	UF : 0, UT : 1,
	J1=   180.000 deg,	J2=   162.834 deg
};
P[215]{
   GP1:
	UF : 1, UT : 1,		CONFIG : 'N U T, 0, 0, 0',
	X =   896.264  mm,	Y =   758.406  mm,	Z =   974.529  mm,
	W =    -7.900 deg,	P =    -8.126 deg,	R =    27.442 deg
   GP2:
	UF : 0, UT : 1,
	J1=   180.000 deg,	J2=   162.834 deg
};
P[216]{
   GP1:
	UF : 1, UT : 1,		CONFIG : 'N U T, 0, 0, 0',
	X =   911.962  mm,	Y =   812.527  mm,	Z =   974.203  mm,
	W =    -6.200 deg,	P =    -4.980 deg,	R =    27.272 deg
   GP2:
	UF : 0, UT : 1,
	J1=   180.000 deg,	J2=   162.834 deg
};
P[217]{
   GP1:
	UF : 1, UT : 1,		CONFIG : 'N U T, 0, 0, 0',
	X =   899.176  mm,	Y =   819.284  mm,	Z =  1032.753  mm,
	W =     -.314 deg,	P =    -5.430 deg,	R =    27.373 deg
   GP2:
	UF : 0, UT : 1,
	J1=   180.000 deg,	J2=   162.834 deg
};
P[218]{
   GP1:
	UF : 1, UT : 1,		CONFIG : 'N U T, 0, 0, 0',
	X =   681.420  mm,	Y =   819.284  mm,	Z =  1312.752  mm,
	W =     -.314 deg,	P =    -5.430 deg,	R =    27.373 deg
   GP2:
	UF : 0, UT : 1,
	J1=   180.000 deg,	J2=   162.834 deg
};
P[219]{
   GP1:
	UF : 1, UT : 1,		CONFIG : 'N U B, 0, 0, 0',
	X =   351.047  mm,	Y =     7.833  mm,	Z =  2455.305  mm,
	W =     -.021 deg,	P =   -39.773 deg,	R =      .020 deg
   GP2:
	UF : 0, UT : 1,
	J1=   180.000 deg,	J2=   162.834 deg
};
P[220]{
   GP1:
	UF : 1, UT : 1,
	J1=     1.807 deg,	J2=   -17.141 deg,	J3=    43.457 deg,
	J4=      .157 deg,	J5=   -93.510 deg,	J6=    56.808 deg
   GP2:
	UF : 0, UT : 1,
	J1=    90.000 deg,	J2=   180.000 deg
};
P[221]{
   GP1:
	UF : 1, UT : 1,		CONFIG : 'N U T, 0, 0, 0',
	X =  1964.565  mm,	Y =     4.795  mm,	Z =  1612.445  mm,
	W =   -22.514 deg,	P =    41.901 deg,	R =    74.339 deg
   GP2:
	UF : 0, UT : 1,
	J1=    90.000 deg,	J2=   180.000 deg
};
P[222]{
   GP1:
	UF : 1, UT : 1,		CONFIG : 'N U T, 0, 0, 0',
	X =  2447.368  mm,	Y =    -1.157  mm,	Z =   875.833  mm,
	W =    -2.714 deg,	P =    44.884 deg,	R =    86.165 deg
   GP2:
	UF : 0, UT : 1,
	J1=    90.000 deg,	J2=   180.000 deg
};
P[223]{
   GP1:
	UF : 1, UT : 1,		CONFIG : 'N U T, 0, 0, 0',
	X =  2375.366  mm,	Y =   -75.636  mm,	Z =  1068.010  mm,
	W =    19.551 deg,	P =    -7.021 deg,	R =   -36.488 deg
   GP2:
	UF : 0, UT : 1,
	J1=    90.000 deg,	J2=    90.000 deg
};
P[224]{
   GP1:
	UF : 1, UT : 1,		CONFIG : 'N U T, 0, 0, 0',
	X =  2796.342  mm,	Y =  1429.156  mm,	Z =   -10.421  mm,
	W =      .000 deg,	P =      .000 deg,	R =    23.425 deg
   GP2:
	UF : 0, UT : 1,
	J1=    90.000 deg,	J2=    90.000 deg
};
P[225]{
   GP1:
	UF : 1, UT : 1,		CONFIG : 'N U T, 0, 0, 0',
	X =  2779.723  mm,	Y =  1421.979  mm,	Z =   -21.231  mm,
	W =    -1.266 deg,	P =    -3.105 deg,	R =    23.431 deg
   GP2:
	UF : 0, UT : 1,
	J1=    90.000 deg,	J2=    90.000 deg
};
P[226]{
   GP1:
	UF : 1, UT : 1,		CONFIG : 'N U T, 0, 0, 0',
	X =  2779.964  mm,	Y =  1421.713  mm,	Z =   -21.036  mm,
	W =    -1.330 deg,	P =    -3.122 deg,	R =    23.452 deg
   GP2:
	UF : 0, UT : 1,
	J1=    90.000 deg,	J2=    90.000 deg
};
P[227]{
   GP1:
	UF : 1, UT : 1,		CONFIG : 'N U T, 0, 0, 0',
	X =  2796.342  mm,	Y =  1429.156  mm,	Z =   -10.421  mm,
	W =      .000 deg,	P =      .000 deg,	R =    23.425 deg
   GP2:
	UF : 0, UT : 1,
	J1=    90.000 deg,	J2=    90.000 deg
};
P[228]{
   GP1:
	UF : 1, UT : 1,		CONFIG : 'N U T, 0, 0, 0',
	X =  2796.343  mm,	Y =  1408.935  mm,	Z =   -22.596  mm,
	W =      .000 deg,	P =      .000 deg,	R =    23.425 deg
   GP2:
	UF : 0, UT : 1,
	J1=    90.000 deg,	J2=    90.000 deg
};
P[229]{
   GP1:
	UF : 1, UT : 1,		CONFIG : 'N U T, 0, 0, 0',
	X =  2796.308  mm,	Y =  1408.958  mm,	Z =   -22.720  mm,
	W =      .007 deg,	P =      .005 deg,	R =    23.421 deg
   GP2:
	UF : 0, UT : 1,
	J1=    90.000 deg,	J2=    90.000 deg
};
P[230]{
   GP1:
	UF : 1, UT : 1,		CONFIG : 'N U T, 0, 0, 0',
	X =  2796.342  mm,	Y =  1429.156  mm,	Z =   -10.421  mm,
	W =      .000 deg,	P =      .000 deg,	R =    23.425 deg
   GP2:
	UF : 0, UT : 1,
	J1=    90.000 deg,	J2=    90.000 deg
};
P[231]{
   GP1:
	UF : 1, UT : 1,		CONFIG : 'N U T, 0, 0, 0',
	X =  2851.225  mm,	Y =  1481.272  mm,	Z =   628.377  mm,
	W =    23.286 deg,	P =   -46.577 deg,	R =   -54.612 deg
   GP2:
	UF : 0, UT : 1,
	J1=    90.000 deg,	J2=    80.000 deg
};
P[232]{
   GP1:
	UF : 1, UT : 1,		CONFIG : 'F U T, 0, 0, 0',
	X =  2809.449  mm,	Y = -1512.393  mm,	Z =   661.548  mm,
	W =   -26.535 deg,	P =   -41.775 deg,	R =    57.162 deg
   GP2:
	UF : 0, UT : 1,
	J1=    90.000 deg,	J2=   -80.000 deg
};
P[233]{
   GP1:
	UF : 1, UT : 1,		CONFIG : 'N U T, 0, 0, 0',
	X =  2141.340  mm,	Y =  -438.241  mm,	Z =   417.943  mm,
	W =   -44.721 deg,	P =     4.092 deg,	R =     4.073 deg
   GP2:
	UF : 0, UT : 1,
	J1=    89.999 deg,	J2=      .000 deg
};
P[234]{
   GP1:
	UF : 1, UT : 1,		CONFIG : 'N U T, 0, 0, 0',
	X =  2154.716  mm,	Y =  -437.126  mm,	Z =   420.005  mm,
	W =   -41.090 deg,	P =     3.840 deg,	R =     4.352 deg
   GP2:
	UF : 0, UT : 1,
	J1=    89.999 deg,	J2=      .000 deg
};
P[235]{
   GP1:
	UF : 1, UT : 1,		CONFIG : 'N U T, 0, 0, 0',
	X =  2186.155  mm,	Y =  -439.272  mm,	Z =   417.702  mm,
	W =   -40.983 deg,	P =     3.829 deg,	R =     4.326 deg
   GP2:
	UF : 0, UT : 1,
	J1=    89.999 deg,	J2=      .000 deg
};
P[236]{
   GP1:
	UF : 1, UT : 1,		CONFIG : 'N U T, 0, 0, -1',
	X =  2085.564  mm,	Y =   124.051  mm,	Z =   864.116  mm,
	W =     -.715 deg,	P =    43.124 deg,	R =   157.497 deg
   GP2:
	UF : 0, UT : 1,
	J1=    89.999 deg,	J2=    90.000 deg
};
P[672]{
   GP1:
	UF : 1, UT : 1,		CONFIG : 'N U T, 0, 0, 0',
	X =  2790.143  mm,	Y =    51.223  mm,	Z =   753.259  mm,
	W =   -32.541 deg,	P =    32.747 deg,	R =    40.290 deg
   GP2:
	UF : 0, UT : 1,
	J1=    90.000 deg,	J2=   180.000 deg
};
P[673]{
   GP1:
	UF : 1, UT : 1,		CONFIG : 'N U T, 0, 0, 0',
	X =  2827.690  mm,	Y =    49.321  mm,	Z =   754.374  mm,
	W =   -32.607 deg,	P =    32.790 deg,	R =    40.253 deg
   GP2:
	UF : 0, UT : 1,
	J1=    90.000 deg,	J2=   180.000 deg
};
P[674]{
   GP1:
	UF : 1, UT : 1,		CONFIG : 'N U T, 0, 0, 0',
	X =  2780.720  mm,	Y =    85.310  mm,	Z =   845.034  mm,
	W =   -26.000 deg,	P =    27.653 deg,	R =    43.586 deg
   GP2:
	UF : 0, UT : 1,
	J1=    90.000 deg,	J2=   180.000 deg
};
P[675]{
   GP1:
	UF : 1, UT : 1,		CONFIG : 'N U T, 0, 0, 0',
	X =  2810.125  mm,	Y =   -14.508  mm,	Z =   877.692  mm,
	W =     4.233 deg,	P =     1.150 deg,	R =   -15.151 deg
   GP2:
	UF : 0, UT : 1,
	J1=    90.000 deg,	J2=   180.000 deg
};
P[676]{
   GP1:
	UF : 1, UT : 1,		CONFIG : 'N U T, 0, 0, 0',
	X =  2779.721  mm,	Y =   -75.691  mm,	Z =   818.586  mm,
	W =    22.126 deg,	P =    31.326 deg,	R =   -51.965 deg
   GP2:
	UF : 0, UT : 1,
	J1=    90.000 deg,	J2=   180.000 deg
};
P[677]{
   GP1:
	UF : 1, UT : 1,		CONFIG : 'N U T, 0, 0, 0',
	X =  2792.677  mm,	Y =   -55.688  mm,	Z =   756.492  mm,
	W =    24.186 deg,	P =    33.500 deg,	R =   -50.860 deg
   GP2:
	UF : 0, UT : 1,
	J1=    90.000 deg,	J2=   180.000 deg
};
P[678]{
   GP1:
	UF : 1, UT : 1,		CONFIG : 'N U T, 0, 0, 0',
	X =  2832.302  mm,	Y =   -54.185  mm,	Z =   758.283  mm,
	W =    24.209 deg,	P =    33.526 deg,	R =   -50.852 deg
   GP2:
	UF : 0, UT : 1,
	J1=    90.000 deg,	J2=   180.000 deg
};
P[679]{
   GP1:
	UF : 1, UT : 1,		CONFIG : 'N U T, 0, 0, 0',
	X =  2779.721  mm,	Y =   -75.691  mm,	Z =   876.586  mm,
	W =    23.118 deg,	P =    32.394 deg,	R =   -51.441 deg
   GP2:
	UF : 0, UT : 1,
	J1=    90.000 deg,	J2=   180.000 deg
};
P[680]{
   GP1:
	UF : 1, UT : 1,		CONFIG : 'N U T, 0, 0, 0',
	X =  2779.721  mm,	Y =   -75.691  mm,	Z =   876.586  mm,
	W =     -.000 deg,	P =     6.847 deg,	R =      .007 deg
   GP2:
	UF : 0, UT : 1,
	J1=    90.000 deg,	J2=   180.000 deg
};
P[681]{
   GP1:
	UF : 1, UT : 1,		CONFIG : 'N U T, 0, 0, 0',
	X =  2840.099  mm,	Y =   -54.094  mm,	Z =   811.805  mm,
	W =      .000 deg,	P =    10.475 deg,	R =      .007 deg
   GP2:
	UF : 0, UT : 1,
	J1=    90.000 deg,	J2=   180.000 deg
};
P[682]{
   GP1:
	UF : 1, UT : 1,		CONFIG : 'N U T, 0, 0, 0',
	X =  2840.358  mm,	Y =   -49.439  mm,	Z =   753.835  mm,
	W =      .034 deg,	P =    10.479 deg,	R =      .019 deg
   GP2:
	UF : 0, UT : 1,
	J1=    90.000 deg,	J2=   180.000 deg
};
P[683]{
   GP1:
	UF : 1, UT : 1,		CONFIG : 'N U T, 0, 0, 0',
	X =  2841.066  mm,	Y =    46.936  mm,	Z =   753.793  mm,
	W =      .058 deg,	P =    10.474 deg,	R =      .009 deg
   GP2:
	UF : 0, UT : 1,
	J1=    90.000 deg,	J2=   180.000 deg
};
P[684]{
   GP1:
	UF : 1, UT : 1,		CONFIG : 'N U T, 0, 0, 0',
	X =  2840.099  mm,	Y =   -54.094  mm,	Z =   811.805  mm,
	W =      .000 deg,	P =    10.475 deg,	R =      .007 deg
   GP2:
	UF : 0, UT : 1,
	J1=    90.000 deg,	J2=   180.000 deg
};
P[685]{
   GP1:
	UF : 1, UT : 1,		CONFIG : 'N U T, 0, 0, 0',
	X =  2685.813  mm,	Y =   -54.094  mm,	Z =  1008.948  mm,
	W =     -.002 deg,	P =   -13.112 deg,	R =      .007 deg
   GP2:
	UF : 0, UT : 1,
	J1=    90.000 deg,	J2=   180.000 deg
};
P[686]{
   GP1:
	UF : 1, UT : 1,		CONFIG : 'N U T, 0, 0, 0',
	X =  1792.252  mm,	Y =    19.310  mm,	Z =   722.821  mm,
	W =   -31.232 deg,	P =    38.925 deg,	R =    72.124 deg
   GP2:
	UF : 0, UT : 1,
	J1=    90.000 deg,	J2=   180.000 deg
};
P[687]{
   GP1:
	UF : 1, UT : 1,		CONFIG : 'N U T, 0, 0, 0',
	X =  1696.704  mm,	Y =  -379.767  mm,	Z =   546.319  mm,
	W =     0.000 deg,	P =    43.571 deg,	R =    90.007 deg
   GP2:
	UF : 0, UT : 1,
	J1=    90.000 deg,	J2=   180.000 deg
};
P[688]{
   GP1:
	UF : 1, UT : 1,		CONFIG : 'N U T, 0, 0, 0',
	X =  1720.777  mm,	Y =  -450.296  mm,	Z =   422.624  mm,
	W =     -.005 deg,	P =    43.535 deg,	R =    86.286 deg
   GP2:
	UF : 0, UT : 1,
	J1=    90.000 deg,	J2=   180.000 deg
};
P[689]{
   GP1:
	UF : 1, UT : 1,		CONFIG : 'N U T, 0, 0, 0',
	X =  1580.851  mm,	Y =  -449.343  mm,	Z =   421.313  mm,
	W =     -.007 deg,	P =    43.521 deg,	R =    86.268 deg
   GP2:
	UF : 0, UT : 1,
	J1=    90.000 deg,	J2=   180.000 deg
};
P[690]{
   GP1:
	UF : 1, UT : 1,		CONFIG : 'N U T, 0, 0, 0',
	X =  1587.135  mm,	Y =  -378.521  mm,	Z =   501.393  mm,
	W =      .000 deg,	P =    43.571 deg,	R =    86.288 deg
   GP2:
	UF : 0, UT : 1,
	J1=    90.000 deg,	J2=   180.000 deg
};
P[691]{
   GP1:
	UF : 1, UT : 1,		CONFIG : 'N U T, 0, 0, 0',
	X =  1998.349  mm,	Y =  -373.244  mm,	Z =   510.901  mm,
	W =   -38.646 deg,	P =    21.930 deg,	R =    21.323 deg
   GP2:
	UF : 0, UT : 1,
	J1=    90.000 deg,	J2=   180.000 deg
};
P[692]{
   GP1:
	UF : 1, UT : 1,		CONFIG : 'N U T, 0, 0, 0',
	X =  1957.677  mm,	Y =  -448.116  mm,	Z =   422.495  mm,
	W =   -40.835 deg,	P =    20.797 deg,	R =    22.335 deg
   GP2:
	UF : 0, UT : 1,
	J1=    90.000 deg,	J2=   180.000 deg
};
P[693]{
   GP1:
	UF : 1, UT : 1,		CONFIG : 'N U T, 0, 0, 0',
	X =  2027.930  mm,	Y =  -449.856  mm,	Z =   421.404  mm,
	W =   -43.530 deg,	P =    18.886 deg,	R =    21.391 deg
   GP2:
	UF : 0, UT : 1,
	J1=    90.000 deg,	J2=   180.000 deg
};
P[694]{
   GP1:
	UF : 1, UT : 1,		CONFIG : 'N U T, 0, 0, 0',
	X =  2047.306  mm,	Y =  -108.854  mm,	Z =   590.153  mm,
	W =   -38.646 deg,	P =    21.930 deg,	R =    21.323 deg
   GP2:
	UF : 0, UT : 1,
	J1=    90.000 deg,	J2=   180.000 deg
};
P[695]{
   GP1:
	UF : 1, UT : 1,		CONFIG : 'N U T, 0, 0, 0',
	X =  2053.592  mm,	Y =  -292.854  mm,	Z =   563.211  mm,
	W =   -43.351 deg,	P =    -4.892 deg,	R =    40.339 deg
   GP2:
	UF : 0, UT : 1,
	J1=    90.000 deg,	J2=   180.000 deg
};
P[696]{
   GP1:
	UF : 1, UT : 1,		CONFIG : 'N U T, 0, 0, 0',
	X =  2144.764  mm,	Y =  -384.746  mm,	Z =   419.107  mm,
	W =   -44.891 deg,	P =    -3.592 deg,	R =    39.096 deg
   GP2:
	UF : 0, UT : 1,
	J1=    90.000 deg,	J2=   180.000 deg
};
P[697]{
   GP1:
	UF : 1, UT : 1,		CONFIG : 'N U T, 0, 0, 0',
	X =  2100.455  mm,	Y =  -424.853  mm,	Z =   417.888  mm,
	W =   -43.231 deg,	P =    13.871 deg,	R =    57.009 deg
   GP2:
	UF : 0, UT : 1,
	J1=    89.999 deg,	J2=   180.000 deg
};
P[698]{
   GP1:
	UF : 1, UT : 1,		CONFIG : 'N U T, 0, 0, 0',
	X =  2099.808  mm,	Y =  -430.674  mm,	Z =   419.684  mm,
	W =   -44.233 deg,	P =    -9.263 deg,	R =    60.679 deg
   GP2:
	UF : 0, UT : 1,
	J1=    89.999 deg,	J2=   180.000 deg
};
P[699]{
   GP1:
	UF : 1, UT : 1,		CONFIG : 'N U T, 0, 0, 0',
	X =  2096.561  mm,	Y =  -436.435  mm,	Z =   421.890  mm,
	W =   -46.555 deg,	P =    -2.361 deg,	R =    62.902 deg
   GP2:
	UF : 0, UT : 1,
	J1=    90.000 deg,	J2=   180.000 deg
};
P[700]{
   GP1:
	UF : 1, UT : 1,		CONFIG : 'N U T, 0, 0, 0',
	X =  1980.139  mm,	Y =  -394.363  mm,	Z =   568.863  mm,
	W =   -43.468 deg,	P =    -3.333 deg,	R =    66.484 deg
   GP2:
	UF : 0, UT : 1,
	J1=    90.000 deg,	J2=   180.000 deg
};
P[701]{
   GP1:
	UF : 1, UT : 1,		CONFIG : 'N U T, 0, 0, 0',
	X =  1759.952  mm,	Y =   241.660  mm,	Z =   616.315  mm,
	W =    29.266 deg,	P =    41.264 deg,	R =   -11.299 deg
   GP2:
	UF : 0, UT : 1,
	J1=    90.000 deg,	J2=   180.000 deg
};
P[702]{
   GP1:
	UF : 1, UT : 1,		CONFIG : 'N U T, 0, 0, 0',
	X =  1720.918  mm,	Y =   388.510  mm,	Z =   489.828  mm,
	W =     0.000 deg,	P =    43.571 deg,	R =   -89.993 deg
   GP2:
	UF : 0, UT : 1,
	J1=    90.000 deg,	J2=   180.000 deg
};
P[703]{
   GP1:
	UF : 1, UT : 1,		CONFIG : 'N U T, 0, 0, 0',
	X =  1722.929  mm,	Y =   446.414  mm,	Z =   421.655  mm,
	W =    -1.651 deg,	P =    44.983 deg,	R =   -92.337 deg
   GP2:
	UF : 0, UT : 1,
	J1=    90.000 deg,	J2=   180.000 deg
};
P[704]{
   GP1:
	UF : 1, UT : 1,		CONFIG : 'N U T, 0, 0, 0',
	X =  1584.785  mm,	Y =   445.500  mm,	Z =   419.176  mm,
	W =    -1.657 deg,	P =    45.006 deg,	R =   -92.336 deg
   GP2:
	UF : 0, UT : 1,
	J1=    90.000 deg,	J2=   180.000 deg
};
P[705]{
   GP1:
	UF : 1, UT : 1,		CONFIG : 'N U T, 0, 0, 0',
	X =  1594.524  mm,	Y =   351.963  mm,	Z =   523.980  mm,
	W =      .000 deg,	P =    43.571 deg,	R =   -92.306 deg
   GP2:
	UF : 0, UT : 1,
	J1=    90.000 deg,	J2=   180.000 deg
};
P[706]{
   GP1:
	UF : 1, UT : 1,		CONFIG : 'N U T, 0, 0, 0',
	X =  1972.524  mm,	Y =   351.963  mm,	Z =   523.980  mm,
	W =    31.879 deg,	P =    31.438 deg,	R =   -42.291 deg
   GP2:
	UF : 0, UT : 1,
	J1=    90.000 deg,	J2=   180.000 deg
};
P[707]{
   GP1:
	UF : 1, UT : 1,		CONFIG : 'N U T, 0, 0, 0',
	X =  1957.584  mm,	Y =   447.653  mm,	Z =   420.327  mm,
	W =    32.281 deg,	P =    33.246 deg,	R =   -40.947 deg
   GP2:
	UF : 0, UT : 1,
	J1=    90.000 deg,	J2=   180.000 deg
};
P[708]{
   GP1:
	UF : 1, UT : 1,		CONFIG : 'N U T, 0, 0, 0',
	X =  2031.416  mm,	Y =   447.860  mm,	Z =   420.354  mm,
	W =    34.389 deg,	P =    31.198 deg,	R =   -39.833 deg
   GP2:
	UF : 0, UT : 1,
	J1=    90.000 deg,	J2=   180.000 deg
};
P[709]{
   GP1:
	UF : 1, UT : 1,		CONFIG : 'N U T, 0, 0, 0',
	X =  2028.229  mm,	Y =   306.190  mm,	Z =   574.407  mm,
	W =    39.948 deg,	P =    19.080 deg,	R =   -23.626 deg
   GP2:
	UF : 0, UT : 1,
	J1=    90.000 deg,	J2=   180.000 deg
};
P[710]{
   GP1:
	UF : 1, UT : 1,		CONFIG : 'N U T, 0, 0, 0',
	X =  2028.228  mm,	Y =   306.190  mm,	Z =   574.407  mm,
	W =    39.948 deg,	P =    19.080 deg,	R =   -73.748 deg
   GP2:
	UF : 0, UT : 1,
	J1=    90.000 deg,	J2=   180.000 deg
};
P[711]{
   GP1:
	UF : 1, UT : 1,		CONFIG : 'N U T, 0, 0, 0',
	X =  2146.185  mm,	Y =   382.939  mm,	Z =   421.328  mm,
	W =    42.385 deg,	P =    16.872 deg,	R =   -60.307 deg
   GP2:
	UF : 0, UT : 1,
	J1=    90.000 deg,	J2=   180.000 deg
};
P[712]{
   GP1:
	UF : 1, UT : 1,		CONFIG : 'N U T, 0, 0, 0',
	X =  2104.195  mm,	Y =   420.889  mm,	Z =   422.475  mm,
	W =    44.151 deg,	P =     9.880 deg,	R =   -52.687 deg
   GP2:
	UF : 0, UT : 1,
	J1=    90.000 deg,	J2=   180.000 deg
};
P[713]{
   GP1:
	UF : 1, UT : 1,		CONFIG : 'N U T, 0, 0, 0',
	X =  2101.951  mm,	Y =   428.282  mm,	Z =   420.792  mm,
	W =    44.777 deg,	P =    -5.046 deg,	R =   -67.249 deg
   GP2:
	UF : 0, UT : 1,
	J1=    89.999 deg,	J2=   180.000 deg
};
P[714]{
   GP1:
	UF : 1, UT : 1,		CONFIG : 'N U T, 0, 0, 0',
	X =  2101.615  mm,	Y =   433.364  mm,	Z =   421.849  mm,
	W =    42.053 deg,	P =   -17.708 deg,	R =   -50.532 deg
   GP2:
	UF : 0, UT : 1,
	J1=    89.999 deg,	J2=   180.000 deg
};
P[715]{
   GP1:
	UF : 1, UT : 1,		CONFIG : 'N U T, 0, 0, 0',
	X =  2002.025  mm,	Y =   135.053  mm,	Z =   547.724  mm,
	W =    43.132 deg,	P =    -6.887 deg,	R =   -61.237 deg
   GP2:
	UF : 0, UT : 1,
	J1=    90.000 deg,	J2=   180.000 deg
};
P[716]{
   GP1:
	UF : 1, UT : 1,		CONFIG : 'N U T, 0, 0, 0',
	X =  2377.025  mm,	Y =   240.053  mm,	Z =   291.724  mm,
	W =    40.241 deg,	P =    18.349 deg,	R =   -20.268 deg
   GP2:
	UF : 0, UT : 1,
	J1=    90.000 deg,	J2=   180.000 deg
};
P[717]{
   GP1:
	UF : 1, UT : 1,		CONFIG : 'N U T, 0, 0, 0',
	X =  2355.551  mm,	Y =   374.115  mm,	Z =   302.484  mm,
	W =    40.241 deg,	P =    18.349 deg,	R =   -20.268 deg
   GP2:
	UF : 0, UT : 1,
	J1=    90.000 deg,	J2=   180.000 deg
};
P[718]{
   GP1:
	UF : 1, UT : 1,		CONFIG : 'N U T, 0, 0, 0',
	X =  2349.451  mm,	Y =   438.430  mm,	Z =   272.108  mm,
	W =    44.913 deg,	P =     3.071 deg,	R =    -3.074 deg
   GP2:
	UF : 0, UT : 1,
	J1=    90.000 deg,	J2=   180.000 deg
};
P[719]{
   GP1:
	UF : 1, UT : 1,		CONFIG : 'N U T, 0, 0, 0',
	X =  2407.584  mm,	Y =   438.337  mm,	Z =   273.841  mm,
	W =    38.958 deg,	P =   -20.279 deg,	R =    -1.908 deg
   GP2:
	UF : 0, UT : 1,
	J1=    89.999 deg,	J2=   180.000 deg
};
P[720]{
   GP1:
	UF : 1, UT : 1,		CONFIG : 'N U T, 0, 0, 0',
	X =  2355.551  mm,	Y =   374.115  mm,	Z =   302.484  mm,
	W =    40.241 deg,	P =    18.349 deg,	R =   -20.268 deg
   GP2:
	UF : 0, UT : 1,
	J1=    90.000 deg,	J2=   180.000 deg
};
P[721]{
   GP1:
	UF : 1, UT : 1,		CONFIG : 'N U T, 0, 0, 0',
	X =  2355.551  mm,	Y =   222.115  mm,	Z =   302.484  mm,
	W =    40.242 deg,	P =    18.350 deg,	R =   -20.267 deg
   GP2:
	UF : 0, UT : 1,
	J1=    90.000 deg,	J2=   180.000 deg
};
P[722]{
   GP1:
	UF : 1, UT : 1,		CONFIG : 'N U T, 0, 0, 0',
	X =  2484.503  mm,	Y =   222.115  mm,	Z =   302.484  mm,
	W =    43.394 deg,	P =    -4.399 deg,	R =     4.775 deg
   GP2:
	UF : 0, UT : 1,
	J1=    90.000 deg,	J2=   180.000 deg
};
P[723]{
   GP1:
	UF : 1, UT : 1,		CONFIG : 'N U T, 0, 0, 0',
	X =  2484.503  mm,	Y =   285.115  mm,	Z =   258.737  mm,
	W =    43.394 deg,	P =    -4.398 deg,	R =     4.776 deg
   GP2:
	UF : 0, UT : 1,
	J1=    90.000 deg,	J2=   180.000 deg
};
P[724]{
   GP1:
	UF : 1, UT : 1,		CONFIG : 'N U T, 0, 0, 0',
	X =  2482.396  mm,	Y =   435.010  mm,	Z =   224.036  mm,
	W =     9.249 deg,	P =   -44.227 deg,	R =    76.876 deg
   GP2:
	UF : 0, UT : 1,
	J1=    90.000 deg,	J2=   180.000 deg
};
P[725]{
   GP1:
	UF : 1, UT : 1,		CONFIG : 'N U T, 0, 0, 0',
	X =  2430.889  mm,	Y =   433.696  mm,	Z =   223.972  mm,
	W =    35.355 deg,	P =   -42.180 deg,	R =    70.882 deg
   GP2:
	UF : 0, UT : 1,
	J1=    90.000 deg,	J2=   180.000 deg
};
P[726]{
   GP1:
	UF : 1, UT : 1,		CONFIG : 'N U T, 0, 0, 0',
	X =  2484.503  mm,	Y =   285.115  mm,	Z =   258.737  mm,
	W =    43.394 deg,	P =    -4.398 deg,	R =     4.776 deg
   GP2:
	UF : 0, UT : 1,
	J1=    90.000 deg,	J2=   180.000 deg
};
P[727]{
   GP1:
	UF : 1, UT : 1,		CONFIG : 'N U T, 0, 0, 0',
	X =  2484.503  mm,	Y =   222.115  mm,	Z =   302.485  mm,
	W =    43.394 deg,	P =    -4.399 deg,	R =     4.775 deg
   GP2:
	UF : 0, UT : 1,
	J1=    90.000 deg,	J2=   180.000 deg
};
P[728]{
   GP1:
	UF : 1, UT : 1,		CONFIG : 'N U T, 0, 0, 0',
	X =  2355.551  mm,	Y =     2.115  mm,	Z =   302.485  mm,
	W =     5.759 deg,	P =    43.266 deg,	R =    98.508 deg
   GP2:
	UF : 0, UT : 1,
	J1=    90.000 deg,	J2=   180.000 deg
};
P[729]{
   GP1:
	UF : 1, UT : 1,		CONFIG : 'N U T, 0, 0, 0',
	X =  2355.551  mm,	Y =  -363.653  mm,	Z =   302.484  mm,
	W =   -43.559 deg,	P =     1.197 deg,	R =     1.395 deg
   GP2:
	UF : 0, UT : 1,
	J1=    90.000 deg,	J2=   180.000 deg
};
P[730]{
   GP1:
	UF : 1, UT : 1,		CONFIG : 'N U T, 0, 0, 0',
	X =  2346.935  mm,	Y =  -439.624  mm,	Z =   272.632  mm,
	W =   -44.978 deg,	P =     1.293 deg,	R =     1.297 deg
   GP2:
	UF : 0, UT : 1,
	J1=    90.000 deg,	J2=   180.000 deg
};
P[731]{
   GP1:
	UF : 1, UT : 1,		CONFIG : 'N U T, 0, 0, 0',
	X =  2407.646  mm,	Y =  -437.669  mm,	Z =   274.279  mm,
	W =   -45.256 deg,	P =   -24.481 deg,	R =     5.929 deg
   GP2:
	UF : 0, UT : 1,
	J1=    89.999 deg,	J2=   180.000 deg
};
P[732]{
   GP1:
	UF : 1, UT : 1,		CONFIG : 'N U T, 0, 0, 0',
	X =  2355.551  mm,	Y =  -363.653  mm,	Z =   302.484  mm,
	W =   -43.559 deg,	P =     1.197 deg,	R =     1.395 deg
   GP2:
	UF : 0, UT : 1,
	J1=    90.000 deg,	J2=   180.000 deg
};
P[733]{
   GP1:
	UF : 1, UT : 1,		CONFIG : 'N U T, 0, 0, 0',
	X =  2355.551  mm,	Y =  -226.653  mm,	Z =   302.484  mm,
	W =   -43.560 deg,	P =     1.197 deg,	R =     1.395 deg
   GP2:
	UF : 0, UT : 1,
	J1=    90.000 deg,	J2=   180.000 deg
};
P[734]{
   GP1:
	UF : 1, UT : 1,		CONFIG : 'N U T, 0, 0, 0',
	X =  2475.388  mm,	Y =  -226.653  mm,	Z =   302.484  mm,
	W =   -29.446 deg,	P =   -33.698 deg,	R =   -44.366 deg
   GP2:
	UF : 0, UT : 1,
	J1=    90.000 deg,	J2=   180.000 deg
};
P[735]{
   GP1:
	UF : 1, UT : 1,		CONFIG : 'N U T, 0, 0, 0',
	X =  2484.256  mm,	Y =  -439.439  mm,	Z =   222.852  mm,
	W =    -2.387 deg,	P =   -44.924 deg,	R =   -86.621 deg
   GP2:
	UF : 0, UT : 1,
	J1=    90.000 deg,	J2=   180.000 deg
};
P[736]{
   GP1:
	UF : 1, UT : 1,		CONFIG : 'N U T, 0, 0, 0',
	X =  2426.375  mm,	Y =  -437.302  mm,	Z =   225.413  mm,
	W =   -26.791 deg,	P =   -43.570 deg,	R =   -86.675 deg
   GP2:
	UF : 0, UT : 1,
	J1=    90.000 deg,	J2=   180.000 deg
};
P[737]{
   GP1:
	UF : 1, UT : 1,		CONFIG : 'N U T, 0, 0, 0',
	X =  2475.389  mm,	Y =  -226.653  mm,	Z =   302.484  mm,
	W =   -29.446 deg,	P =   -33.698 deg,	R =   -44.366 deg
   GP2:
	UF : 0, UT : 1,
	J1=    90.000 deg,	J2=   180.000 deg
};
P[738]{
   GP1:
	UF : 1, UT : 1,		CONFIG : 'N U T, 0, 0, 0',
	X =  2475.361  mm,	Y =  -127.379  mm,	Z =   161.610  mm,
	W =    -9.376 deg,	P =    15.683 deg,	R =   -16.267 deg
   GP2:
	UF : 0, UT : 1,
	J1=    90.000 deg,	J2=   180.000 deg
};
P[739]{
   GP1:
	UF : 1, UT : 1,		CONFIG : 'N U T, 0, 0, 0',
	X =  2184.132  mm,	Y =   -42.626  mm,	Z =   871.946  mm,
	W =    -9.375 deg,	P =    15.689 deg,	R =   -16.266 deg
   GP2:
	UF : 0, UT : 1,
	J1=    90.000 deg,	J2=   180.000 deg
};
P[740]{
   GP1:
	UF : 1, UT : 1,		CONFIG : 'N U B, 0, 0, 0',
	X =   390.614  mm,	Y =     -.024  mm,	Z =  2434.016  mm,
	W =     -.021 deg,	P =   -39.773 deg,	R =      .020 deg
   GP2:
	UF : 0, UT : 1,
	J1=    90.000 deg,	J2=   180.000 deg
};
P[741]{
   GP1:
	UF : 1, UT : 1,
	J1=     -.065 deg,	J2=   -43.813 deg,	J3=    64.455 deg,
	J4=     -.068 deg,	J5=   -69.455 deg,	J6=      .029 deg
   GP2:
	UF : 0, UT : 1,
	J1=    90.000 deg,	J2=     0.000 deg
};
P[742]{
   GP1:
	UF : 1, UT : 1,		CONFIG : 'N U T, 0, 0, 0',
	X =  1852.631  mm,	Y =    -6.774  mm,	Z =   565.209  mm,
	W =     -.000 deg,	P =    45.917 deg,	R =    -2.669 deg
   GP2:
	UF : 0, UT : 1,
	J1=    90.000 deg,	J2=     0.000 deg
};
P[743]{
   GP1:
	UF : 1, UT : 1,		CONFIG : 'N U T, 0, 0, 0',
	X =  1655.504  mm,	Y =   141.226  mm,	Z =   511.209  mm,
	W =     -.000 deg,	P =    45.917 deg,	R =    -2.669 deg
   GP2:
	UF : 0, UT : 1,
	J1=    90.000 deg,	J2=     0.000 deg
};
P[744]{
   GP1:
	UF : 1, UT : 1,		CONFIG : 'N U T, 0, 0, 0',
	X =  1609.671  mm,	Y =   144.502  mm,	Z =   412.787  mm,
	W =      .173 deg,	P =    45.931 deg,	R =    -2.572 deg
   GP2:
	UF : 0, UT : 1,
	J1=    90.000 deg,	J2=     -.000 deg
};
P[745]{
   GP1:
	UF : 1, UT : 1,		CONFIG : 'N U T, 0, 0, 0',
	X =  1610.947  mm,	Y =   248.052  mm,	Z =   413.254  mm,
	W =      .102 deg,	P =    45.934 deg,	R =    -2.609 deg
   GP2:
	UF : 0, UT : 1,
	J1=    89.999 deg,	J2=      .000 deg
};
P[746]{
   GP1:
	UF : 1, UT : 1,		CONFIG : 'N U T, 0, 0, 0',
	X =  1637.136  mm,	Y =   314.793  mm,	Z =   459.534  mm,
	W =     -.000 deg,	P =    45.917 deg,	R =    -2.669 deg
   GP2:
	UF : 0, UT : 1,
	J1=    90.000 deg,	J2=     0.000 deg
};
P[747]{
   GP1:
	UF : 1, UT : 1,		CONFIG : 'N U T, 0, 0, 0',
	X =  1612.461  mm,	Y =   348.792  mm,	Z =   411.820  mm,
	W =    -2.031 deg,	P =    48.815 deg,	R =    -2.770 deg
   GP2:
	UF : 0, UT : 1,
	J1=    89.999 deg,	J2=      .000 deg
};
P[748]{
   GP1:
	UF : 1, UT : 1,		CONFIG : 'N U T, 0, 0, 0',
	X =  1610.257  mm,	Y =   432.690  mm,	Z =   411.364  mm,
	W =    32.767 deg,	P =    34.177 deg,	R =    46.223 deg
   GP2:
	UF : 0, UT : 1,
	J1=    90.000 deg,	J2=      .000 deg
};
P[749]{
   GP1:
	UF : 1, UT : 1,		CONFIG : 'N U T, 0, 0, 0',
	X =  1691.137  mm,	Y =   314.793  mm,	Z =   549.534  mm,
	W =     -.000 deg,	P =    45.918 deg,	R =    -2.669 deg
   GP2:
	UF : 0, UT : 1,
	J1=    90.000 deg,	J2=     0.000 deg
};
P[750]{
   GP1:
	UF : 1, UT : 1,		CONFIG : 'N U T, 0, 0, 0',
	X =  1691.136  mm,	Y =  -139.207  mm,	Z =   549.534  mm,
	W =     -.000 deg,	P =    45.919 deg,	R =    -2.669 deg
   GP2:
	UF : 0, UT : 1,
	J1=    90.000 deg,	J2=     0.000 deg
};
P[751]{
   GP1:
	UF : 1, UT : 1,		CONFIG : 'N U T, 0, 0, 0',
	X =  1611.466  mm,	Y =  -130.160  mm,	Z =   407.191  mm,
	W =      .132 deg,	P =    45.900 deg,	R =    -2.610 deg
   GP2:
	UF : 0, UT : 1,
	J1=    89.999 deg,	J2=      .000 deg
};
P[752]{
   GP1:
	UF : 1, UT : 1,		CONFIG : 'N U T, 0, 0, 0',
	X =  1612.455  mm,	Y =  -157.655  mm,	Z =   408.458  mm,
	W =      .071 deg,	P =    45.910 deg,	R =    -2.628 deg
   GP2:
	UF : 0, UT : 1,
	J1=    90.000 deg,	J2=      .000 deg
};
P[753]{
   GP1:
	UF : 1, UT : 1,		CONFIG : 'N U T, 0, 0, 0',
	X =  1701.553  mm,	Y =  -162.044  mm,	Z =   513.926  mm,
	W =      .001 deg,	P =    45.916 deg,	R =    -2.666 deg
   GP2:
	UF : 0, UT : 1,
	J1=    90.000 deg,	J2=     0.000 deg
};
P[754]{
   GP1:
	UF : 1, UT : 1,		CONFIG : 'N U T, 0, 0, 0',
	X =  1651.458  mm,	Y =  -207.923  mm,	Z =   466.756  mm,
	W =      .001 deg,	P =    45.916 deg,	R =    15.512 deg
   GP2:
	UF : 0, UT : 1,
	J1=    90.000 deg,	J2=     0.000 deg
};
P[755]{
   GP1:
	UF : 1, UT : 1,		CONFIG : 'N U T, 0, 0, 0',
	X =  1611.664  mm,	Y =  -223.720  mm,	Z =   410.590  mm,
	W =    -1.058 deg,	P =    39.466 deg,	R =    14.834 deg
   GP2:
	UF : 0, UT : 1,
	J1=    90.000 deg,	J2=      .000 deg
};
P[756]{
   GP1:
	UF : 1, UT : 1,		CONFIG : 'N U T, 0, 0, 0',
	X =  1613.255  mm,	Y =  -156.646  mm,	Z =   408.642  mm,
	W =     3.854 deg,	P =    34.718 deg,	R =   -21.298 deg
   GP2:
	UF : 0, UT : 1,
	J1=    90.000 deg,	J2=      .000 deg
};
P[757]{
   GP1:
	UF : 1, UT : 1,		CONFIG : 'N U T, 0, 0, 0',
	X =  1663.438  mm,	Y =  -190.775  mm,	Z =   486.236  mm,
	W =      .001 deg,	P =    45.916 deg,	R =   -32.606 deg
   GP2:
	UF : 0, UT : 1,
	J1=    90.000 deg,	J2=     0.000 deg
};
P[758]{
   GP1:
	UF : 1, UT : 1,		CONFIG : 'N U T, 0, 0, 0',
	X =  1694.246  mm,	Y =  -335.221  mm,	Z =   519.016  mm,
	W =   -24.937 deg,	P =    39.897 deg,	R =   -38.608 deg
   GP2:
	UF : 0, UT : 1,
	J1=    90.000 deg,	J2=     0.000 deg
};
P[759]{
   GP1:
	UF : 1, UT : 1,		CONFIG : 'N U T, 0, 0, 0',
	X =  1609.958  mm,	Y =  -354.596  mm,	Z =   409.981  mm,
	W =   -28.732 deg,	P =    41.555 deg,	R =   -39.650 deg
   GP2:
	UF : 0, UT : 1,
	J1=    90.000 deg,	J2=      .000 deg
};
P[760]{
   GP1:
	UF : 1, UT : 1,		CONFIG : 'N U T, 0, 0, 0',
	X =  1607.480  mm,	Y =  -434.366  mm,	Z =   408.044  mm,
	W =   -34.474 deg,	P =    37.257 deg,	R =   -48.669 deg
   GP2:
	UF : 0, UT : 1,
	J1=    90.000 deg,	J2=      .000 deg
};
P[761]{
   GP1:
	UF : 1, UT : 1,		CONFIG : 'N U T, 0, 0, 0',
	X =  1714.229  mm,	Y =  -410.520  mm,	Z =   541.553  mm,
	W =   -30.592 deg,	P =    36.083 deg,	R =   -32.808 deg
   GP2:
	UF : 0, UT : 1,
	J1=    90.000 deg,	J2=     0.000 deg
};
P[762]{
   GP1:
	UF : 1, UT : 1,		CONFIG : 'N U T, 0, 0, 0',
	X =  1852.631  mm,	Y =    -6.774  mm,	Z =   565.209  mm,
	W =     -.000 deg,	P =    45.917 deg,	R =    -2.669 deg
   GP2:
	UF : 0, UT : 1,
	J1=    90.000 deg,	J2=     0.000 deg
};
P[763]{
   GP1:
	UF : 1, UT : 1,		CONFIG : 'N U T, 0, 0, 0',
	X =  2052.631  mm,	Y =  -276.774  mm,	Z =   565.209  mm,
	W =   -41.084 deg,	P =    22.633 deg,	R =    21.147 deg
   GP2:
	UF : 0, UT : 1,
	J1=    90.000 deg,	J2=     0.000 deg
};
P[764]{
   GP1:
	UF : 1, UT : 1,		CONFIG : 'N U T, 0, 0, 0',
	X =  2088.553  mm,	Y =  -373.284  mm,	Z =   491.208  mm,
	W =   -45.800 deg,	P =     3.716 deg,	R =      .937 deg
   GP2:
	UF : 0, UT : 1,
	J1=    90.000 deg,	J2=     0.000 deg
};
P[765]{
   GP1:
	UF : 1, UT : 1,		CONFIG : 'N U T, 0, 0, 0',
	X =  2063.471  mm,	Y =  -440.130  mm,	Z =   414.294  mm,
	W =   -44.841 deg,	P =     4.112 deg,	R =     4.121 deg
   GP2:
	UF : 0, UT : 1,
	J1=    90.000 deg,	J2=      .000 deg
};
P[766]{
   GP1:
	UF : 1, UT : 1,		CONFIG : 'N U T, 0, 0, 0',
	X =  2311.826  mm,	Y =  -442.485  mm,	Z =   415.387  mm,
	W =   -44.797 deg,	P =     4.102 deg,	R =     4.097 deg
   GP2:
	UF : 0, UT : 1,
	J1=    89.999 deg,	J2=      .000 deg
};
P[767]{
   GP1:
	UF : 1, UT : 1,		CONFIG : 'N U T, 0, 0, 0',
	X =  2305.976  mm,	Y =  -368.534  mm,	Z =   500.330  mm,
	W =   -45.801 deg,	P =     3.717 deg,	R =     4.521 deg
   GP2:
	UF : 0, UT : 1,
	J1=    90.000 deg,	J2=     0.000 deg
};
P[768]{
   GP1:
	UF : 1, UT : 1,		CONFIG : 'N U T, 0, 0, 0',
	X =  2315.872  mm,	Y =  -419.741  mm,	Z =   406.098  mm,
	W =   -44.926 deg,	P =     1.424 deg,	R =    -8.822 deg
   GP2:
	UF : 0, UT : 1,
	J1=    90.000 deg,	J2=      .000 deg
};
P[769]{
   GP1:
	UF : 1, UT : 1,		CONFIG : 'N U T, 0, 0, 0',
	X =  2238.454  mm,	Y =  -405.307  mm,	Z =   405.845  mm,
	W =   -44.909 deg,	P =     2.942 deg,	R =   -10.342 deg
   GP2:
	UF : 0, UT : 1,
	J1=    89.999 deg,	J2=      .000 deg
};
P[770]{
   GP1:
	UF : 1, UT : 1,		CONFIG : 'N U T, 0, 0, 0',
	X =  2163.271  mm,	Y =  -384.781  mm,	Z =   405.753  mm,
	W =   -44.753 deg,	P =      .541 deg,	R =   -16.094 deg
   GP2:
	UF : 0, UT : 1,
	J1=    89.999 deg,	J2=      .000 deg
};
P[771]{
   GP1:
	UF : 1, UT : 1,		CONFIG : 'N U T, 0, 0, 0',
	X =  2185.243  mm,	Y =  -309.879  mm,	Z =   500.265  mm,
	W =   -45.800 deg,	P =     3.717 deg,	R =   -19.293 deg
   GP2:
	UF : 0, UT : 1,
	J1=    90.000 deg,	J2=     0.000 deg
};
P[772]{
   GP1:
	UF : 1, UT : 1,		CONFIG : 'N U T, 0, 0, 0',
	X =  2354.243  mm,	Y =  -309.879  mm,	Z =   717.265  mm,
	W =   -45.800 deg,	P =     3.717 deg,	R =     3.840 deg
   GP2:
	UF : 0, UT : 1,
	J1=    90.000 deg,	J2=     0.000 deg
};
P[773]{
   GP1:
	UF : 1, UT : 1,		CONFIG : 'N U T, 0, 0, 0',
	X =  2342.588  mm,	Y =  -441.901  mm,	Z =   567.316  mm,
	W =   -44.855 deg,	P =     3.773 deg,	R =     3.782 deg
   GP2:
	UF : 0, UT : 1,
	J1=    90.000 deg,	J2=      .000 deg
};
P[774]{
   GP1:
	UF : 1, UT : 1,		CONFIG : 'N U T, 0, 0, 0',
	X =  2403.136  mm,	Y =  -439.944  mm,	Z =   567.175  mm,
	W =   -49.121 deg,	P =     -.390 deg,	R =    21.519 deg
   GP2:
	UF : 0, UT : 1,
	J1=    89.999 deg,	J2=      .000 deg
};
P[775]{
   GP1:
	UF : 1, UT : 1,		CONFIG : 'N U T, 0, 0, 0',
	X =  2354.243  mm,	Y =  -309.879  mm,	Z =   717.265  mm,
	W =   -45.800 deg,	P =     3.717 deg,	R =     3.840 deg
   GP2:
	UF : 0, UT : 1,
	J1=    90.000 deg,	J2=     0.000 deg
};
P[776]{
   GP1:
	UF : 1, UT : 1,		CONFIG : 'N U T, 0, 0, 0',
	X =  2424.155  mm,	Y =  -399.247  mm,	Z =   717.265  mm,
	W =   -45.800 deg,	P =     3.717 deg,	R =     3.840 deg
   GP2:
	UF : 0, UT : 1,
	J1=    90.000 deg,	J2=     0.000 deg
};
P[777]{
   GP1:
	UF : 1, UT : 1,		CONFIG : 'N U T, 0, 0, 0',
	X =  2482.618  mm,	Y =  -440.224  mm,	Z =   618.446  mm,
	W =   -44.879 deg,	P =     3.779 deg,	R =     3.789 deg
   GP2:
	UF : 0, UT : 1,
	J1=    90.000 deg,	J2=      .000 deg
};
P[778]{
   GP1:
	UF : 1, UT : 1,		CONFIG : 'N U T, 0, 0, 0',
	X =  2426.441  mm,	Y =  -440.765  mm,	Z =   617.885  mm,
	W =   -44.875 deg,	P =     3.774 deg,	R =     3.782 deg
   GP2:
	UF : 0, UT : 1,
	J1=    90.000 deg,	J2=     0.000 deg
};
P[779]{
   GP1:
	UF : 1, UT : 1,		CONFIG : 'N U T, 0, 0, 0',
	X =  2422.927  mm,	Y =  -439.786  mm,	Z =   619.638  mm,
	W =   -47.202 deg,	P =    -4.228 deg,	R =    12.058 deg
   GP2:
	UF : 0, UT : 1,
	J1=    90.000 deg,	J2=     0.000 deg
};
P[780]{
   GP1:
	UF : 1, UT : 1,		CONFIG : 'N U T, 0, 0, 0',
	X =  2412.831  mm,	Y =  -438.608  mm,	Z =   617.946  mm,
	W =   -54.100 deg,	P =   -12.118 deg,	R =    21.734 deg
   GP2:
	UF : 0, UT : 1,
	J1=    90.000 deg,	J2=      .000 deg
};
P[781]{
   GP1:
	UF : 1, UT : 1,		CONFIG : 'N U T, 0, 0, 0',
	X =  2474.892  mm,	Y =  -236.857  mm,	Z =   699.878  mm,
	W =   -45.800 deg,	P =     3.717 deg,	R =     3.840 deg
   GP2:
	UF : 0, UT : 1,
	J1=    90.000 deg,	J2=     0.000 deg
};
P[782]{
   GP1:
	UF : 1, UT : 1,		CONFIG : 'N U T, 0, 0, 0',
	X =  2498.018  mm,	Y =  -347.318  mm,	Z =   570.880  mm,
	W =   -28.620 deg,	P =   -37.578 deg,	R =   -47.947 deg
   GP2:
	UF : 0, UT : 1,
	J1=    90.000 deg,	J2=     0.000 deg
};
P[783]{
   GP1:
	UF : 1, UT : 1,		CONFIG : 'N U T, 0, 0, 0',
	X =  2483.026  mm,	Y =  -442.881  mm,	Z =   516.609  mm,
	W =     -.757 deg,	P =   -44.978 deg,	R =   -88.928 deg
   GP2:
	UF : 0, UT : 1,
	J1=    90.000 deg,	J2=      .000 deg
};
P[784]{
   GP1:
	UF : 1, UT : 1,		CONFIG : 'N U T, 0, 0, 0',
	X =  2425.172  mm,	Y =  -441.096  mm,	Z =   516.929  mm,
	W =   -46.015 deg,	P =   -32.689 deg,	R =   -60.060 deg
   GP2:
	UF : 0, UT : 1,
	J1=    90.000 deg,	J2=      .000 deg
};
P[785]{
   GP1:
	UF : 1, UT : 1,		CONFIG : 'N U T, 0, 0, 0',
	X =  2560.160  mm,	Y =  -368.783  mm,	Z =   604.364  mm,
	W =   -28.619 deg,	P =   -37.577 deg,	R =   -73.349 deg
   GP2:
	UF : 0, UT : 1,
	J1=    90.000 deg,	J2=     0.000 deg
};
P[786]{
   GP1:
	UF : 1, UT : 1,		CONFIG : 'N U T, 0, 0, 0',
	X =  2560.160  mm,	Y =  -188.783  mm,	Z =   604.364  mm,
	W =   -28.619 deg,	P =   -37.577 deg,	R =   -18.464 deg
   GP2:
	UF : 0, UT : 1,
	J1=    90.000 deg,	J2=     0.000 deg
};
P[787]{
   GP1:
	UF : 1, UT : 1,		CONFIG : 'N U T, 0, 0, 0',
	X =  2065.242  mm,	Y =   379.121  mm,	Z =   528.266  mm,
	W =    43.428 deg,	P =    16.677 deg,	R =   -20.967 deg
   GP2:
	UF : 0, UT : 1,
	J1=    90.000 deg,	J2=     0.000 deg
};
P[788]{
   GP1:
	UF : 1, UT : 1,		CONFIG : 'N U T, 0, 0, 0',
	X =  2063.097  mm,	Y =   437.980  mm,	Z =   414.739  mm,
	W =    42.297 deg,	P =    17.060 deg,	R =   -17.870 deg
   GP2:
	UF : 0, UT : 1,
	J1=    90.000 deg,	J2=      .000 deg
};
P[789]{
   GP1:
	UF : 1, UT : 1,		CONFIG : 'N U T, 0, 0, 0',
	X =  2316.160  mm,	Y =   435.659  mm,	Z =   417.388  mm,
	W =    42.299 deg,	P =    17.065 deg,	R =   -17.871 deg
   GP2:
	UF : 0, UT : 1,
	J1=    90.000 deg,	J2=      .000 deg
};
P[790]{
   GP1:
	UF : 1, UT : 1,		CONFIG : 'N U T, 0, 0, 0',
	X =  2302.760  mm,	Y =   370.627  mm,	Z =   499.650  mm,
	W =    43.428 deg,	P =    16.677 deg,	R =   -18.246 deg
   GP2:
	UF : 0, UT : 1,
	J1=    90.000 deg,	J2=     0.000 deg
};
P[791]{
   GP1:
	UF : 1, UT : 1,		CONFIG : 'N U T, 0, 0, 0',
	X =  2315.088  mm,	Y =   415.032  mm,	Z =   410.831  mm,
	W =    34.268 deg,	P =    15.906 deg,	R =    -9.927 deg
   GP2:
	UF : 0, UT : 1,
	J1=    90.000 deg,	J2=      .000 deg
};
P[792]{
   GP1:
	UF : 1, UT : 1,		CONFIG : 'N U T, 0, 0, 0',
	X =  2233.834  mm,	Y =   395.684  mm,	Z =   410.334  mm,
	W =    42.564 deg,	P =    16.228 deg,	R =    -3.478 deg
   GP2:
	UF : 0, UT : 1,
	J1=    90.000 deg,	J2=      .000 deg
};
P[793]{
   GP1:
	UF : 1, UT : 1,		CONFIG : 'N U T, 0, 0, 0',
	X =  2159.172  mm,	Y =   379.102  mm,	Z =   406.936  mm,
	W =    42.409 deg,	P =    16.706 deg,	R =     -.973 deg
   GP2:
	UF : 0, UT : 1,
	J1=    90.000 deg,	J2=      .000 deg
};
P[794]{
   GP1:
	UF : 1, UT : 1,		CONFIG : 'N U T, 0, 0, 0',
	X =  2175.664  mm,	Y =   307.835  mm,	Z =   684.697  mm,
	W =    43.428 deg,	P =    16.677 deg,	R =    -1.009 deg
   GP2:
	UF : 0, UT : 1,
	J1=    90.000 deg,	J2=     0.000 deg
};
P[795]{
   GP1:
	UF : 1, UT : 1,		CONFIG : 'N U T, 0, 0, 0',
	X =  2352.664  mm,	Y =   365.835  mm,	Z =   684.697  mm,
	W =    43.428 deg,	P =    16.677 deg,	R =   -16.431 deg
   GP2:
	UF : 0, UT : 1,
	J1=    90.000 deg,	J2=     0.000 deg
};
P[796]{
   GP1:
	UF : 1, UT : 1,		CONFIG : 'N U T, 0, 0, 0',
	X =  2345.371  mm,	Y =   435.818  mm,	Z =   568.431  mm,
	W =    42.336 deg,	P =    16.930 deg,	R =   -17.720 deg
   GP2:
	UF : 0, UT : 1,
	J1=    90.000 deg,	J2=      .000 deg
};
P[797]{
   GP1:
	UF : 1, UT : 1,		CONFIG : 'N U T, 0, 0, 0',
	X =  2402.616  mm,	Y =   434.310  mm,	Z =   568.239  mm,
	W =    45.526 deg,	P =      .647 deg,	R =   -34.327 deg
   GP2:
	UF : 0, UT : 1,
	J1=    89.999 deg,	J2=      .000 deg
};
P[798]{
   GP1:
	UF : 1, UT : 1,		CONFIG : 'N U T, 0, 0, 0',
	X =  2352.664  mm,	Y =   365.835  mm,	Z =   684.697  mm,
	W =    43.428 deg,	P =    16.677 deg,	R =   -18.155 deg
   GP2:
	UF : 0, UT : 1,
	J1=    90.000 deg,	J2=     0.000 deg
};
P[799]{
   GP1:
	UF : 1, UT : 1,		CONFIG : 'N U T, 0, 0, 0',
	X =  2483.065  mm,	Y =   435.633  mm,	Z =   619.433  mm,
	W =    42.329 deg,	P =    17.028 deg,	R =   -17.828 deg
   GP2:
	UF : 0, UT : 1,
	J1=    90.000 deg,	J2=      .000 deg
};
P[800]{
   GP1:
	UF : 1, UT : 1,		CONFIG : 'N U T, 0, 0, 0',
	X =  2428.112  mm,	Y =   434.137  mm,	Z =   619.473  mm,
	W =    42.315 deg,	P =    17.019 deg,	R =   -17.826 deg
   GP2:
	UF : 0, UT : 1,
	J1=    90.000 deg,	J2=      .000 deg
};
P[801]{
   GP1:
	UF : 1, UT : 1,		CONFIG : 'N U T, 0, 0, 0',
	X =  2418.833  mm,	Y =   433.862  mm,	Z =   619.119  mm,
	W =    49.444 deg,	P =     7.080 deg,	R =   -20.554 deg
   GP2:
	UF : 0, UT : 1,
	J1=    90.000 deg,	J2=      .000 deg
};
P[802]{
   GP1:
	UF : 1, UT : 1,		CONFIG : 'N U T, 0, 0, 0',
	X =  2411.050  mm,	Y =   432.026  mm,	Z =   615.794  mm,
	W =    55.585 deg,	P =     -.624 deg,	R =   -30.576 deg
   GP2:
	UF : 0, UT : 1,
	J1=    90.000 deg,	J2=     0.000 deg
};
P[803]{
   GP1:
	UF : 1, UT : 1,		CONFIG : 'N U T, 0, 0, 0',
	X =  2496.124  mm,	Y =   220.970  mm,	Z =   706.785  mm,
	W =    43.428 deg,	P =    16.677 deg,	R =   -18.155 deg
   GP2:
	UF : 0, UT : 1,
	J1=    90.000 deg,	J2=     0.000 deg
};
P[804]{
   GP1:
	UF : 1, UT : 1,		CONFIG : 'N U T, 0, 0, 0',
	X =  2496.124  mm,	Y =   371.970  mm,	Z =   564.784  mm,
	W =    28.310 deg,	P =   -37.796 deg,	R =    47.397 deg
   GP2:
	UF : 0, UT : 1,
	J1=    90.000 deg,	J2=     0.000 deg
};
P[805]{
   GP1:
	UF : 1, UT : 1,		CONFIG : 'N U T, 0, 0, 0',
	X =  2481.086  mm,	Y =   435.399  mm,	Z =   517.416  mm,
	W =    -2.570 deg,	P =   -44.922 deg,	R =    93.655 deg
   GP2:
	UF : 0, UT : 1,
	J1=    90.000 deg,	J2=      .000 deg
};
P[806]{
   GP1:
	UF : 1, UT : 1,		CONFIG : 'N U T, 0, 0, 0',
	X =  2425.311  mm,	Y =   433.891  mm,	Z =   519.254  mm,
	W =    33.691 deg,	P =   -40.561 deg,	R =    68.577 deg
   GP2:
	UF : 0, UT : 1,
	J1=    90.000 deg,	J2=      .000 deg
};
P[807]{
   GP1:
	UF : 1, UT : 1,		CONFIG : 'N U T, 0, 0, 0',
	X =  2505.724  mm,	Y =   371.970  mm,	Z =   545.104  mm,
	W =    28.310 deg,	P =   -37.796 deg,	R =    47.397 deg
   GP2:
	UF : 0, UT : 1,
	J1=    90.000 deg,	J2=     0.000 deg
};
P[808]{
   GP1:
	UF : 1, UT : 1,		CONFIG : 'N U T, 0, 0, 0',
	X =  2496.124  mm,	Y =    40.970  mm,	Z =   706.786  mm,
	W =    43.428 deg,	P =    16.677 deg,	R =   -18.155 deg
   GP2:
	UF : 0, UT : 1,
	J1=    90.000 deg,	J2=     0.000 deg
};
P[809]{
   GP1:
	UF : 1, UT : 1,		CONFIG : 'N U T, 0, 0, 0',
	X =  1825.123  mm,	Y =    84.024  mm,	Z =   706.785  mm,
	W =    -6.286 deg,	P =    45.581 deg,	R =  -100.055 deg
   GP2:
	UF : 0, UT : 1,
	J1=    90.000 deg,	J2=     0.000 deg
};
P[810]{
   GP1:
	UF : 1, UT : 1,		CONFIG : 'N U B, 0, 0, 0',
	X =   390.614  mm,	Y =     -.024  mm,	Z =  2434.016  mm,
	W =     -.021 deg,	P =   -39.773 deg,	R =      .020 deg
   GP2:
	UF : 0, UT : 1,
	J1=    90.000 deg,	J2=     0.000 deg
};
P[811]{
   GP1:
	UF : 1, UT : 1,		CONFIG : 'N U T, 0, 0, 0',
	X =  1169.761  mm,	Y =  1400.668  mm,	Z =  1377.270  mm,
	W =     2.123 deg,	P =   -27.834 deg,	R =    46.073 deg
   GP2:
	UF : 0, UT : 1,
	J1=    90.000 deg,	J2=    90.000 deg
};
P[812]{
   GP1:
	UF : 1, UT : 1,		CONFIG : 'N U T, 0, 0, 0',
	X =  2160.560  mm,	Y =  1340.283  mm,	Z =   479.513  mm,
	W =     3.095 deg,	P =    -8.630 deg,	R =    30.802 deg
   GP2:
	UF : 0, UT : 1,
	J1=    90.000 deg,	J2=    90.000 deg
};
P[813]{
   GP1:
	UF : 1, UT : 1,		CONFIG : 'N U T, 0, 0, 0',
	X =  2796.342  mm,	Y =  1419.988  mm,	Z =    24.239  mm,
	W =      .000 deg,	P =      .000 deg,	R =    23.425 deg
   GP2:
	UF : 0, UT : 1,
	J1=    90.000 deg,	J2=    90.000 deg
};
P[814]{
   GP1:
	UF : 1, UT : 1,		CONFIG : 'N U T, 0, 0, 0',
	X =  2796.240  mm,	Y =  1434.830  mm,	Z =   -20.868  mm,
	W =    -1.935 deg,	P =    -4.569 deg,	R =    23.477 deg
   GP2:
	UF : 0, UT : 1,
	J1=    90.000 deg,	J2=    90.000 deg
};
P[815]{
   GP1:
	UF : 1, UT : 1,		CONFIG : 'N U T, 0, 0, 0',
	X =  2796.240  mm,	Y =  1434.830  mm,	Z =   -20.868  mm,
	W =    -1.935 deg,	P =    -4.569 deg,	R =    23.477 deg
   GP2:
	UF : 0, UT : 1,
	J1=    90.000 deg,	J2=    90.000 deg
};
P[816]{
   GP1:
	UF : 1, UT : 1,		CONFIG : 'N U T, 0, 0, 0',
	X =  2796.342  mm,	Y =  1434.707  mm,	Z =    58.334  mm,
	W =      .000 deg,	P =      .000 deg,	R =    23.425 deg
   GP2:
	UF : 0, UT : 1,
	J1=    90.000 deg,	J2=    90.000 deg
};
P[817]{
   GP1:
	UF : 1, UT : 1,		CONFIG : 'N U T, 0, 0, 0',
	X =  2379.579  mm,	Y =  1303.563  mm,	Z =   243.935  mm,
	W =   -10.292 deg,	P =     3.753 deg,	R =    25.430 deg
   GP2:
	UF : 0, UT : 1,
	J1=    90.000 deg,	J2=    90.000 deg
};
P[818]{
   GP1:
	UF : 1, UT : 1,		CONFIG : 'N U T, 0, 0, 0',
	X =  1425.741  mm,	Y =   537.295  mm,	Z =   426.307  mm,
	W =   -37.512 deg,	P =    -9.236 deg,	R =    21.393 deg
   GP2:
	UF : 0, UT : 1,
	J1=    90.000 deg,	J2=    90.000 deg
};
P[819]{
   GP1:
	UF : 1, UT : 1,		CONFIG : 'N U T, 0, 0, 0',
	X =  1439.456  mm,	Y =   227.579  mm,	Z =    82.897  mm,
	W =   -43.796 deg,	P =    -2.383 deg,	R =    15.668 deg
   GP2:
	UF : 0, UT : 1,
	J1=    90.000 deg,	J2=    90.000 deg
};
P[820]{
   GP1:
	UF : 1, UT : 1,
	J1=    12.170 deg,	J2=   -42.804 deg,	J3=   -24.846 deg,
	J4=    75.067 deg,	J5=   -27.353 deg,	J6=   -37.008 deg
   GP2:
	UF : 0, UT : 1,
	J1=    90.000 deg,	J2=    90.000 deg
};
P[821]{
   GP1:
	UF : 1, UT : 1,
	J1=    10.193 deg,	J2=   -38.006 deg,	J3=   -29.309 deg,
	J4=    82.275 deg,	J5=   -30.701 deg,	J6=   -47.783 deg
   GP2:
	UF : 0, UT : 1,
	J1=    90.000 deg,	J2=    90.000 deg
};
P[822]{
   GP1:
	UF : 1, UT : 1,		CONFIG : 'N U T, 0, 0, 0',
	X =  1483.187  mm,	Y =   -32.092  mm,	Z =   -42.652  mm,
	W =   -44.722 deg,	P =     5.497 deg,	R =    17.517 deg
   GP2:
	UF : 0, UT : 1,
	J1=    90.000 deg,	J2=    90.000 deg
};
P[823]{
   GP1:
	UF : 1, UT : 1,		CONFIG : 'N U T, 0, 0, 0',
	X =  1498.238  mm,	Y =   -27.378  mm,	Z =   -40.373  mm,
	W =   -44.733 deg,	P =     5.508 deg,	R =    32.342 deg
   GP2:
	UF : 0, UT : 1,
	J1=    90.000 deg,	J2=    90.000 deg
};
P[824]{
   GP1:
	UF : 1, UT : 1,		CONFIG : 'N U T, 0, 0, 0',
	X =  1504.966  mm,	Y =   -16.747  mm,	Z =   -39.003  mm,
	W =   -44.734 deg,	P =     5.503 deg,	R =    65.609 deg
   GP2:
	UF : 0, UT : 1,
	J1=    90.000 deg,	J2=    90.000 deg
};
P[825]{
   GP1:
	UF : 1, UT : 1,		CONFIG : 'N U T, 0, 0, 0',
	X =  1511.354  mm,	Y =    32.208  mm,	Z =   -37.699  mm,
	W =   -36.293 deg,	P =   -28.673 deg,	R =    51.824 deg
   GP2:
	UF : 0, UT : 1,
	J1=    90.000 deg,	J2=    90.000 deg
};
P[826]{
   GP1:
	UF : 1, UT : 1,		CONFIG : 'N U T, 0, 0, 0',
	X =  1524.743  mm,	Y =    52.776  mm,	Z =   -40.640  mm,
	W =   -30.310 deg,	P =    34.943 deg,	R =    61.025 deg
   GP2:
	UF : 0, UT : 1,
	J1=    90.000 deg,	J2=    90.000 deg
};
P[827]{
   GP1:
	UF : 1, UT : 1,		CONFIG : 'N U T, 0, 0, 0',
	X =  1546.251  mm,	Y =    47.295  mm,	Z =   -42.912  mm,
	W =   -44.969 deg,	P =    -1.364 deg,	R =   -46.388 deg
   GP2:
	UF : 0, UT : 1,
	J1=    90.000 deg,	J2=    90.000 deg
};
P[828]{
   GP1:
	UF : 1, UT : 1,		CONFIG : 'N U T, 0, 0, 0',
	X =  1576.609  mm,	Y =    13.312  mm,	Z =   -45.161  mm,
	W =   -44.972 deg,	P =    -1.331 deg,	R =   -46.412 deg
   GP2:
	UF : 0, UT : 1,
	J1=    90.000 deg,	J2=    90.000 deg
};
P[829]{
   GP1:
	UF : 1, UT : 1,		CONFIG : 'N U T, 0, 0, 0',
	X =  1584.799  mm,	Y =     8.317  mm,	Z =   -43.206  mm,
	W =   -44.959 deg,	P =    -1.326 deg,	R =   -46.409 deg
   GP2:
	UF : 0, UT : 1,
	J1=    90.000 deg,	J2=    90.000 deg
};
P[830]{
   GP1:
	UF : 1, UT : 1,		CONFIG : 'N U T, 0, 0, 0',
	X =  1595.851  mm,	Y =   168.471  mm,	Z =    12.234  mm,
	W =   -43.745 deg,	P =    -3.325 deg,	R =    -4.329 deg
   GP2:
	UF : 0, UT : 1,
	J1=    90.000 deg,	J2=    90.000 deg
};
P[831]{
   GP1:
	UF : 1, UT : 1,		CONFIG : 'N U T, 0, 0, 0',
	X =  1790.704  mm,	Y =   213.074  mm,	Z =    23.022  mm,
	W =    50.484 deg,	P =     5.553 deg,	R =   -78.853 deg
   GP2:
	UF : 0, UT : 1,
	J1=    90.000 deg,	J2=    90.000 deg
};
P[832]{
   GP1:
	UF : 1, UT : 1,		CONFIG : 'N U T, 0, 0, 0',
	X =  1934.971  mm,	Y =    90.847  mm,	Z =    21.992  mm,
	W =    44.321 deg,	P =     6.701 deg,	R =   -79.548 deg
   GP2:
	UF : 0, UT : 1,
	J1=    90.000 deg,	J2=    90.000 deg
};
P[833]{
   GP1:
	UF : 1, UT : 1,		CONFIG : 'N U T, 0, 0, 0',
	X =  2032.099  mm,	Y =    33.450  mm,	Z =   -38.212  mm,
	W =    40.098 deg,	P =    22.435 deg,	R =  -114.326 deg
   GP2:
	UF : 0, UT : 1,
	J1=    89.999 deg,	J2=    90.000 deg
};
P[834]{
   GP1:
	UF : 1, UT : 1,		CONFIG : 'N U T, 0, 0, -1',
	X =  2049.069  mm,	Y =     9.346  mm,	Z =   -34.789  mm,
	W =    48.817 deg,	P =    10.905 deg,	R =  -129.577 deg
   GP2:
	UF : 0, UT : 1,
	J1=    89.999 deg,	J2=    90.000 deg
};
P[835]{
   GP1:
	UF : 1, UT : 1,		CONFIG : 'N U T, 0, 0, 0',
	X =  1879.866  mm,	Y =   103.962  mm,	Z =    68.602  mm,
	W =    32.019 deg,	P =    14.952 deg,	R =  -129.625 deg
   GP2:
	UF : 0, UT : 1,
	J1=    90.000 deg,	J2=    90.000 deg
};
P[842]{
   GP1:
	UF : 1, UT : 1,		CONFIG : 'N U T, 0, 0, 0',
	X =   689.476  mm,	Y =   450.392  mm,	Z =    80.587  mm,
	W =    -2.211 deg,	P =    43.411 deg,	R =   -86.182 deg
   GP2:
	UF : 0, UT : 1,
	J1=    90.000 deg,	J2=    90.000 deg
};
P[843]{
   GP1:
	UF : 1, UT : 1,		CONFIG : 'N U T, 0, 0, 0',
	X =  1250.850  mm,	Y =  -232.930  mm,	Z =    12.233  mm,
	W =    33.676 deg,	P =    29.929 deg,	R =    49.697 deg
   GP2:
	UF : 0, UT : 1,
	J1=    90.000 deg,	J2=    90.000 deg
};
P[844]{
   GP1:
	UF : 1, UT : 1,		CONFIG : 'N U T, 0, 0, 0',
	X =  1783.851  mm,	Y =  -338.130  mm,	Z =    12.233  mm,
	W =    33.676 deg,	P =    29.929 deg,	R =    49.697 deg
   GP2:
	UF : 0, UT : 1,
	J1=    90.000 deg,	J2=    90.000 deg
};
P[845]{
   GP1:
	UF : 1, UT : 1,		CONFIG : 'N U T, 0, 0, 0',
	X =  1679.271  mm,	Y =  -490.428  mm,	Z =   -42.534  mm,
	W =     5.231 deg,	P =    44.768 deg,	R =    15.413 deg
   GP2:
	UF : 0, UT : 1,
	J1=    90.000 deg,	J2=    90.000 deg
};
P[846]{
   GP1:
	UF : 1, UT : 1,		CONFIG : 'N U T, 0, 0, 0',
	X =  1614.266  mm,	Y =   -29.526  mm,	Z =   -42.280  mm,
	W =    37.974 deg,	P =    26.237 deg,	R =    68.462 deg
   GP2:
	UF : 0, UT : 1,
	J1=    90.000 deg,	J2=    90.000 deg
};
P[847]{
   GP1:
	UF : 1, UT : 1,		CONFIG : 'N U T, 0, 0, 0',
	X =  1685.335  mm,	Y =   -60.794  mm,	Z =    56.902  mm,
	W =    41.445 deg,	P =    15.816 deg,	R =    46.464 deg
   GP2:
	UF : 0, UT : 1,
	J1=    90.000 deg,	J2=    90.000 deg
};
P[848]{
   GP1:
	UF : 1, UT : 1,		CONFIG : 'N U T, 0, 0, 0',
	X =  1913.446  mm,	Y =   -62.657  mm,	Z =   130.915  mm,
	W =   -26.067 deg,	P =   -28.164 deg,	R =    87.762 deg
   GP2:
	UF : 0, UT : 1,
	J1=    75.000 deg,	J2=    90.000 deg
};
P[849]{
   GP1:
	UF : 1, UT : 1,		CONFIG : 'N U T, 0, 0, 0',
	X =  1955.399  mm,	Y =   -13.539  mm,	Z =    38.320  mm,
	W =   -20.495 deg,	P =   -27.294 deg,	R =    86.815 deg
   GP2:
	UF : 0, UT : 1,
	J1=    75.000 deg,	J2=    90.000 deg
};
P[850]{
   GP1:
	UF : 1, UT : 1,		CONFIG : 'N U T, 0, 0, 0',
	X =  1993.467  mm,	Y =   -68.392  mm,	Z =    26.636  mm,
	W =   -14.672 deg,	P =   -26.883 deg,	R =    84.191 deg
   GP2:
	UF : 0, UT : 1,
	J1=    75.000 deg,	J2=    90.000 deg
};
P[851]{
   GP1:
	UF : 1, UT : 1,		CONFIG : 'N U T, 0, 0, 0',
	X =  2010.541  mm,	Y =   -94.243  mm,	Z =    22.582  mm,
	W =   -14.675 deg,	P =   -26.885 deg,	R =    84.189 deg
   GP2:
	UF : 0, UT : 1,
	J1=    75.000 deg,	J2=    90.000 deg
};
P[852]{
   GP1:
	UF : 1, UT : 1,		CONFIG : 'N U T, 0, 0, 0',
	X =  2023.206  mm,	Y =  -114.415  mm,	Z =    18.237  mm,
	W =   -19.566 deg,	P =   -27.930 deg,	R =    84.815 deg
   GP2:
	UF : 0, UT : 1,
	J1=    75.000 deg,	J2=    90.000 deg
};
P[853]{
   GP1:
	UF : 1, UT : 1,		CONFIG : 'N U T, 0, 0, 0',
	X =  2039.378  mm,	Y =  -135.448  mm,	Z =    13.382  mm,
	W =   -13.820 deg,	P =   -36.350 deg,	R =    95.180 deg
   GP2:
	UF : 0, UT : 1,
	J1=    75.000 deg,	J2=    90.000 deg
};
P[854]{
   GP1:
	UF : 1, UT : 1,		CONFIG : 'N U T, 0, 0, 0',
	X =  2054.566  mm,	Y =  -142.905  mm,	Z =     8.414  mm,
	W =    -3.677 deg,	P =   -40.350 deg,	R =    86.323 deg
   GP2:
	UF : 0, UT : 1,
	J1=    75.000 deg,	J2=    90.000 deg
};
P[855]{
   GP1:
	UF : 1, UT : 1,		CONFIG : 'N U T, 0, 0, 0',
	X =  2127.986  mm,	Y =  -179.204  mm,	Z =    -8.471  mm,
	W =    -1.490 deg,	P =   -40.478 deg,	R =    83.072 deg
   GP2:
	UF : 0, UT : 1,
	J1=    75.000 deg,	J2=    90.000 deg
};
P[856]{
   GP1:
	UF : 1, UT : 1,		CONFIG : 'N U T, 0, 0, 0',
	X =  2154.020  mm,	Y =  -196.097  mm,	Z =   -14.879  mm,
	W =    -8.355 deg,	P =   -36.865 deg,	R =    82.663 deg
   GP2:
	UF : 0, UT : 1,
	J1=    75.000 deg,	J2=    90.000 deg
};
P[857]{
   GP1:
	UF : 1, UT : 1,		CONFIG : 'N U T, 0, 0, 0',
	X =  2299.027  mm,	Y =  -303.490  mm,	Z =   -51.207  mm,
	W =    20.582 deg,	P =   -32.263 deg,	R =    33.785 deg
   GP2:
	UF : 0, UT : 1,
	J1=    75.000 deg,	J2=    90.000 deg
};
P[858]{
   GP1:
	UF : 1, UT : 1,		CONFIG : 'N U T, 0, 0, 0',
	X =  2329.946  mm,	Y =  -335.417  mm,	Z =   -60.024  mm,
	W =   -26.408 deg,	P =   -19.640 deg,	R =    95.166 deg
   GP2:
	UF : 0, UT : 1,
	J1=    75.000 deg,	J2=    90.000 deg
};
P[859]{
   GP1:
	UF : 1, UT : 1,		CONFIG : 'N U T, 0, 0, 0',
	X =  2341.098  mm,	Y =  -380.731  mm,	Z =   -64.593  mm,
	W =   -29.910 deg,	P =    -2.402 deg,	R =    85.826 deg
   GP2:
	UF : 0, UT : 1,
	J1=    75.000 deg,	J2=    90.000 deg
};
P[860]{
   GP1:
	UF : 1, UT : 1,		CONFIG : 'N U T, 0, 0, 0',
	X =  2340.662  mm,	Y =  -533.390  mm,	Z =   -64.104  mm,
	W =   -26.091 deg,	P =   -15.348 deg,	R =    61.586 deg
   GP2:
	UF : 0, UT : 1,
	J1=    75.000 deg,	J2=    90.000 deg
};
P[861]{
   GP1:
	UF : 1, UT : 1,		CONFIG : 'N U T, 0, 0, 0',
	X =  2365.150  mm,	Y =  -567.969  mm,	Z =   -68.744  mm,
	W =    44.921 deg,	P =     -.806 deg,	R =     8.102 deg
   GP2:
	UF : 0, UT : 1,
	J1=    75.000 deg,	J2=    90.000 deg
};
P[862]{
   GP1:
	UF : 1, UT : 1,		CONFIG : 'N U T, 0, 0, 0',
	X =  2409.481  mm,	Y =  -546.147  mm,	Z =   -86.786  mm,
	W =    53.375 deg,	P =    29.924 deg,	R =    49.281 deg
   GP2:
	UF : 0, UT : 1,
	J1=    75.000 deg,	J2=    90.000 deg
};
P[863]{
   GP1:
	UF : 1, UT : 1,		CONFIG : 'N U T, 0, 0, 0',
	X =  2459.813  mm,	Y =  -506.183  mm,	Z =   -97.056  mm,
	W =    44.281 deg,	P =   -15.560 deg,	R =    28.105 deg
   GP2:
	UF : 0, UT : 1,
	J1=    75.000 deg,	J2=    90.000 deg
};
P[864]{
   GP1:
	UF : 1, UT : 1,		CONFIG : 'N U T, 0, 0, 0',
	X =  2530.042  mm,	Y =  -577.464  mm,	Z =  -112.605  mm,
	W =   -19.567 deg,	P =   -23.190 deg,	R =    42.062 deg
   GP2:
	UF : 0, UT : 1,
	J1=    75.000 deg,	J2=    90.000 deg
};
P[865]{
   GP1:
	UF : 1, UT : 1,		CONFIG : 'N U T, 0, 0, 0',
	X =  2528.068  mm,	Y =  -899.653  mm,	Z =  -111.809  mm,
	W =   -24.862 deg,	P =   -17.327 deg,	R =    57.273 deg
   GP2:
	UF : 0, UT : 1,
	J1=    75.000 deg,	J2=    90.000 deg
};
P[866]{
   GP1:
	UF : 1, UT : 1,		CONFIG : 'N U T, 0, 0, 0',
	X =  2430.793  mm,	Y =  -903.370  mm,	Z =   103.434  mm,
	W =   -23.326 deg,	P =   -26.866 deg,	R =    43.658 deg
   GP2:
	UF : 0, UT : 1,
	J1=    75.000 deg,	J2=    90.000 deg
};
P[867]{
   GP1:
	UF : 1, UT : 1,		CONFIG : 'N U T, 0, 0, 0',
	X =  2368.792  mm,	Y = -1104.074  mm,	Z =    14.434  mm,
	W =   -23.326 deg,	P =   -26.866 deg,	R =    43.658 deg
   GP2:
	UF : 0, UT : 1,
	J1=    75.000 deg,	J2=    90.000 deg
};
P[868]{
   GP1:
	UF : 1, UT : 1,		CONFIG : 'N U T, 0, 0, 0',
	X =  2406.610  mm,	Y = -1082.928  mm,	Z =   -79.092  mm,
	W =   -19.546 deg,	P =   -23.191 deg,	R =    42.044 deg
   GP2:
	UF : 0, UT : 1,
	J1=    75.000 deg,	J2=    90.000 deg
};
P[869]{
   GP1:
	UF : 1, UT : 1,		CONFIG : 'N U T, 0, 0, 0',
	X =  2406.240  mm,	Y = -1067.454  mm,	Z =   -79.890  mm,
	W =   -26.072 deg,	P =   -15.376 deg,	R =    61.548 deg
   GP2:
	UF : 0, UT : 1,
	J1=    75.000 deg,	J2=    90.000 deg
};
P[870]{
   GP1:
	UF : 1, UT : 1,		CONFIG : 'N U T, 0, 0, 0',
	X =  2411.328  mm,	Y = -1059.339  mm,	Z =   -82.122  mm,
	W =   -29.529 deg,	P =     5.502 deg,	R =    57.417 deg
   GP2:
	UF : 0, UT : 1,
	J1=    75.000 deg,	J2=    90.000 deg
};
P[871]{
   GP1:
	UF : 1, UT : 1,		CONFIG : 'N U T, 0, 0, 0',
	X =  2417.737  mm,	Y = -1058.858  mm,	Z =   -87.317  mm,
	W =   -32.089 deg,	P =    36.210 deg,	R =    28.759 deg
   GP2:
	UF : 0, UT : 1,
	J1=    75.000 deg,	J2=    90.000 deg
};
P[872]{
   GP1:
	UF : 1, UT : 1,		CONFIG : 'N U T, 0, 0, 0',
	X =  2433.460  mm,	Y = -1056.417  mm,	Z =   -89.488  mm,
	W =   -32.089 deg,	P =    36.208 deg,	R =    28.755 deg
   GP2:
	UF : 0, UT : 1,
	J1=    75.000 deg,	J2=    90.000 deg
};
P[873]{
   GP1:
	UF : 1, UT : 1,		CONFIG : 'N U T, 0, 0, 0',
	X =  2490.094  mm,	Y = -1043.948  mm,	Z =  -104.256  mm,
	W =   -34.501 deg,	P =    16.016 deg,	R =    43.409 deg
   GP2:
	UF : 0, UT : 1,
	J1=    75.000 deg,	J2=    90.000 deg
};
P[874]{
   GP1:
	UF : 1, UT : 1,		CONFIG : 'N U T, 0, 0, 0',
	X =  2516.545  mm,	Y = -1011.556  mm,	Z =  -109.379  mm,
	W =   -31.920 deg,	P =     -.640 deg,	R =    54.341 deg
   GP2:
	UF : 0, UT : 1,
	J1=    75.000 deg,	J2=    90.000 deg
};
P[875]{
   GP1:
	UF : 1, UT : 1,		CONFIG : 'N U T, 0, 0, 0',
	X =  2527.383  mm,	Y =  -994.955  mm,	Z =  -113.224  mm,
	W =   -33.554 deg,	P =     6.843 deg,	R =    49.559 deg
   GP2:
	UF : 0, UT : 1,
	J1=    75.000 deg,	J2=    90.000 deg
};
P[876]{
   GP1:
	UF : 1, UT : 1,		CONFIG : 'N U T, 0, 0, 0',
	X =  2539.741  mm,	Y =  -971.323  mm,	Z =  -114.238  mm,
	W =   -29.429 deg,	P =    -8.196 deg,	R =    58.724 deg
   GP2:
	UF : 0, UT : 1,
	J1=    75.000 deg,	J2=    90.000 deg
};
P[877]{
   GP1:
	UF : 1, UT : 1,		CONFIG : 'N U T, 0, 0, 0',
	X =  2534.996  mm,	Y =  -932.454  mm,	Z =  -113.004  mm,
	W =   -16.664 deg,	P =   -27.549 deg,	R =    67.339 deg
   GP2:
	UF : 0, UT : 1,
	J1=    75.000 deg,	J2=    90.000 deg
};
P[878]{
   GP1:
	UF : 1, UT : 1,		CONFIG : 'N U T, 0, 0, 0',
	X =  2530.050  mm,	Y =  -916.394  mm,	Z =  -110.772  mm,
	W =   -21.954 deg,	P =   -21.718 deg,	R =    65.079 deg
   GP2:
	UF : 0, UT : 1,
	J1=    75.000 deg,	J2=    90.000 deg
};
P[879]{
   GP1:
	UF : 1, UT : 1,		CONFIG : 'N U T, 0, 0, 0',
	X =  2527.190  mm,	Y =  -898.692  mm,	Z =  -109.493  mm,
	W =   -26.202 deg,	P =   -15.169 deg,	R =    61.996 deg
   GP2:
	UF : 0, UT : 1,
	J1=    75.000 deg,	J2=    90.000 deg
};
P[880]{
   GP1:
	UF : 1, UT : 1,		CONFIG : 'N U T, 0, 0, 1',
	X =  2343.611  mm,	Y =  -907.396  mm,	Z =   140.307  mm,
	W =   -59.893 deg,	P =   -10.052 deg,	R =    84.220 deg
   GP2:
	UF : 0, UT : 1,
	J1=    75.000 deg,	J2=    90.000 deg
};
P[881]{
   GP1:
	UF : 1, UT : 1,		CONFIG : 'N U T, 0, 0, 0',
	X =  1150.634  mm,	Y =  -892.054  mm,	Z =   818.818  mm,
	W =   -59.893 deg,	P =   -10.052 deg,	R =    84.220 deg
   GP2:
	UF : 0, UT : 1,
	J1=    80.000 deg,	J2=    90.000 deg
};
P[882]{
   GP1:
	UF : 1, UT : 1,		CONFIG : 'N U T, 0, 0, 0',
	X =   521.831  mm,	Y = -1015.927  mm,	Z =   836.270  mm,
	W =    -8.786 deg,	P =    50.997 deg,	R =    66.144 deg
   GP2:
	UF : 0, UT : 1,
	J1=    80.000 deg,	J2=    90.000 deg
};
P[883]{
   GP1:
	UF : 1, UT : 1,		CONFIG : 'N U T, 0, 0, 0',
	X =   710.644  mm,	Y =     3.965  mm,	Z =  1496.074  mm,
	W =   -24.135 deg,	P =    23.300 deg,	R =    55.066 deg
   GP2:
	UF : 0, UT : 1,
	J1=    80.000 deg,	J2=    90.000 deg
};
P[884]{
   GP1:
	UF : 1, UT : 1,		CONFIG : 'N U T, 0, 0, -1',
	X =  2063.024  mm,	Y =   140.025  mm,	Z =   970.779  mm,
	W =    -3.034 deg,	P =    45.241 deg,	R =   165.093 deg
   GP2:
	UF : 0, UT : 1,
	J1=    90.000 deg,	J2=    90.000 deg
};
P[885]{
   GP1:
	UF : 1, UT : 1,		CONFIG : 'N U T, 0, 0, -1',
	X =  2077.801  mm,	Y =   102.634  mm,	Z =   864.459  mm,
	W =     -.693 deg,	P =    43.134 deg,	R =   157.506 deg
   GP2:
	UF : 0, UT : 1,
	J1=    89.999 deg,	J2=    90.000 deg
};
P[886]{
   GP1:
	UF : 1, UT : 1,		CONFIG : 'N U T, 0, 0, 0',
	X =  2075.878  mm,	Y =   148.875  mm,	Z =   863.326  mm,
	W =      .395 deg,	P =    43.419 deg,	R =  -114.443 deg
   GP2:
	UF : 0, UT : 1,
	J1=    89.999 deg,	J2=    90.000 deg
};
P[887]{
   GP1:
	UF : 1, UT : 1,		CONFIG : 'N U T, 0, 0, 0',
	X =  2047.235  mm,	Y =   141.441  mm,	Z =   862.686  mm,
	W =      .266 deg,	P =    43.290 deg,	R =   -16.093 deg
   GP2:
	UF : 0, UT : 1,
	J1=    90.000 deg,	J2=    90.000 deg
};
P[888]{
   GP1:
	UF : 1, UT : 1,		CONFIG : 'N U T, 0, 0, 0',
	X =  2032.386  mm,	Y =    94.306  mm,	Z =   863.797  mm,
	W =     -.955 deg,	P =    43.088 deg,	R =   -19.865 deg
   GP2:
	UF : 0, UT : 1,
	J1=    89.999 deg,	J2=    90.000 deg
};
P[889]{
   GP1:
	UF : 1, UT : 1,		CONFIG : 'N U T, 0, 0, 0',
	X =  2045.852  mm,	Y =    71.656  mm,	Z =   862.184  mm,
	W =      .985 deg,	P =    43.307 deg,	R =    72.945 deg
   GP2:
	UF : 0, UT : 1,
	J1=    90.000 deg,	J2=    90.000 deg
};
P[890]{
   GP1:
	UF : 1, UT : 1,		CONFIG : 'N U T, 0, 0, 0',
	X =  2071.666  mm,	Y =    81.698  mm,	Z =   863.376  mm,
	W =      .625 deg,	P =    42.194 deg,	R =   151.061 deg
   GP2:
	UF : 0, UT : 1,
	J1=    90.000 deg,	J2=    90.000 deg
};
P[891]{
   GP1:
	UF : 1, UT : 1,		CONFIG : 'N U T, 0, 0, 0',
	X =  2078.289  mm,	Y =   102.157  mm,	Z =   863.070  mm,
	W =      .142 deg,	P =    42.671 deg,	R =   157.880 deg
   GP2:
	UF : 0, UT : 1,
	J1=    90.000 deg,	J2=    90.000 deg
};
P[892]{
   GP1:
	UF : 1, UT : 1,		CONFIG : 'N U T, 0, 0, 0',
	X =  2049.931  mm,	Y =    77.805  mm,	Z =  1030.403  mm,
	W =     3.803 deg,	P =    43.129 deg,	R =   172.126 deg
   GP2:
	UF : 0, UT : 1,
	J1=    90.000 deg,	J2=    90.000 deg
};
P[893]{
   GP1:
	UF : 1, UT : 1,		CONFIG : 'N U T, 0, 0, 0',
	X =  2090.009  mm,	Y =   205.805  mm,	Z =  1030.403  mm,
	W =    -6.392 deg,	P =    42.881 deg,	R =    76.256 deg
   GP2:
	UF : 0, UT : 1,
	J1=    90.000 deg,	J2=    90.000 deg
};
P[894]{
   GP1:
	UF : 1, UT : 1,		CONFIG : 'N U T, 0, 0, 0',
	X =  2062.519  mm,	Y =   180.497  mm,	Z =   861.554  mm,
	W =    -6.387 deg,	P =    42.873 deg,	R =    81.031 deg
   GP2:
	UF : 0, UT : 1,
	J1=    90.000 deg,	J2=    90.000 deg
};
P[895]{
   GP1:
	UF : 1, UT : 1,		CONFIG : 'N U T, 0, 0, 0',
	X =  2174.520  mm,	Y =   180.106  mm,	Z =   863.074  mm,
	W =    -6.392 deg,	P =    42.881 deg,	R =    81.019 deg
   GP2:
	UF : 0, UT : 1,
	J1=    90.000 deg,	J2=    90.000 deg
};
P[896]{
   GP1:
	UF : 1, UT : 1,		CONFIG : 'N U T, 0, 0, 0',
	X =  2221.599  mm,	Y =   158.867  mm,	Z =   861.206  mm,
	W =    -6.328 deg,	P =    42.856 deg,	R =    37.062 deg
   GP2:
	UF : 0, UT : 1,
	J1=    90.000 deg,	J2=    90.000 deg
};
P[897]{
   GP1:
	UF : 1, UT : 1,		CONFIG : 'N U T, 0, 0, 0',
	X =  2244.893  mm,	Y =   114.757  mm,	Z =   861.492  mm,
	W =    -6.322 deg,	P =    42.884 deg,	R =     2.366 deg
   GP2:
	UF : 0, UT : 1,
	J1=    90.000 deg,	J2=    90.000 deg
};
P[898]{
   GP1:
	UF : 1, UT : 1,		CONFIG : 'N U T, 0, 0, 0',
	X =  2341.485  mm,	Y =   -49.711  mm,	Z =   862.794  mm,
	W =    -6.381 deg,	P =    42.869 deg,	R =    40.648 deg
   GP2:
	UF : 0, UT : 1,
	J1=    90.000 deg,	J2=    90.000 deg
};
P[899]{
   GP1:
	UF : 1, UT : 1,		CONFIG : 'N U T, 0, 0, 0',
	X =  2546.714  mm,	Y =   -99.139  mm,	Z =   864.640  mm,
	W =    -6.392 deg,	P =    42.880 deg,	R =    80.792 deg
   GP2:
	UF : 0, UT : 1,
	J1=    90.000 deg,	J2=    90.000 deg
};
P[900]{
   GP1:
	UF : 1, UT : 1,		CONFIG : 'N U T, 0, 0, 0',
	X =  2596.829  mm,	Y =  -109.510  mm,	Z =   863.742  mm,
	W =   -16.119 deg,	P =    40.648 deg,	R =    47.370 deg
   GP2:
	UF : 0, UT : 1,
	J1=    90.000 deg,	J2=    90.000 deg
};
P[901]{
   GP1:
	UF : 1, UT : 1,		CONFIG : 'N U T, 0, 0, 0',
	X =  2625.885  mm,	Y =  -138.610  mm,	Z =   862.959  mm,
	W =   -32.655 deg,	P =    30.025 deg,	R =    -5.267 deg
   GP2:
	UF : 0, UT : 1,
	J1=    90.000 deg,	J2=    90.000 deg
};
P[902]{
   GP1:
	UF : 1, UT : 1,		CONFIG : 'N U T, 0, 0, 0',
	X =  2647.850  mm,	Y =  -178.137  mm,	Z =   863.251  mm,
	W =   -32.721 deg,	P =    30.015 deg,	R =     -.301 deg
   GP2:
	UF : 0, UT : 1,
	J1=    90.000 deg,	J2=    90.000 deg
};
P[903]{
   GP1:
	UF : 1, UT : 1,		CONFIG : 'N U T, 0, 0, 0',
	X =  2655.688  mm,	Y =  -173.702  mm,	Z =   956.035  mm,
	W =   -32.753 deg,	P =    30.014 deg,	R =    10.111 deg
   GP2:
	UF : 0, UT : 1,
	J1=    90.000 deg,	J2=    90.000 deg
};
P[904]{
   GP1:
	UF : 1, UT : 1,		CONFIG : 'N U T, 0, 0, 0',
	X =  2655.687  mm,	Y =  -345.701  mm,	Z =   956.035  mm,
	W =   -18.106 deg,	P =    33.354 deg,	R =    -8.090 deg
   GP2:
	UF : 0, UT : 1,
	J1=    90.000 deg,	J2=    90.000 deg
};
P[905]{
   GP1:
	UF : 1, UT : 1,		CONFIG : 'N U T, 0, 0, 0',
	X =  2752.136  mm,	Y =  -345.701  mm,	Z =   956.035  mm,
	W =   -15.637 deg,	P =    18.786 deg,	R =    -8.670 deg
   GP2:
	UF : 0, UT : 1,
	J1=    90.000 deg,	J2=    90.000 deg
};
P[906]{
   GP1:
	UF : 1, UT : 1,		CONFIG : 'N U T, 0, 0, 0',
	X =  2651.125  mm,	Y =  -181.965  mm,	Z =   865.326  mm,
	W =     -.409 deg,	P =    36.670 deg,	R =    25.404 deg
   GP2:
	UF : 0, UT : 1,
	J1=    90.000 deg,	J2=    90.000 deg
};
P[907]{
   GP1:
	UF : 1, UT : 1,		CONFIG : 'N U T, 0, 0, 0',
	X =  2712.963  mm,	Y =  -297.527  mm,	Z =   864.372  mm,
	W =   -17.171 deg,	P =    33.307 deg,	R =    -3.589 deg
   GP2:
	UF : 0, UT : 1,
	J1=    90.000 deg,	J2=    90.000 deg
};
P[908]{
   GP1:
	UF : 1, UT : 1,		CONFIG : 'N U T, 0, 0, 0',
	X =  2759.202  mm,	Y =  -384.011  mm,	Z =   866.352  mm,
	W =   -26.306 deg,	P =    25.182 deg,	R =   -22.716 deg
   GP2:
	UF : 0, UT : 1,
	J1=    90.000 deg,	J2=    90.000 deg
};
P[909]{
   GP1:
	UF : 1, UT : 1,		CONFIG : 'N U T, 0, 0, 0',
	X =  2800.634  mm,	Y =  -462.037  mm,	Z =   869.406  mm,
	W =   -35.059 deg,	P =    21.146 deg,	R =   -19.889 deg
   GP2:
	UF : 0, UT : 1,
	J1=    90.000 deg,	J2=    90.000 deg
};
P[910]{
   GP1:
	UF : 1, UT : 1,		CONFIG : 'N U T, 0, 0, 0',
	X =  2864.597  mm,	Y =  -587.463  mm,	Z =   866.155  mm,
	W =   -40.163 deg,	P =    17.500 deg,	R =    -9.073 deg
   GP2:
	UF : 0, UT : 1,
	J1=    90.000 deg,	J2=    90.000 deg
};
P[911]{
   GP1:
	UF : 1, UT : 1,		CONFIG : 'N U T, 0, 0, 0',
	X =  2892.084  mm,	Y =  -550.347  mm,	Z =   921.026  mm,
	W =   -46.061 deg,	P =    13.790 deg,	R =    -1.425 deg
   GP2:
	UF : 0, UT : 1,
	J1=    90.000 deg,	J2=    90.000 deg
};
P[912]{
   GP1:
	UF : 1, UT : 1,		CONFIG : 'N U T, 0, 0, 0',
	X =  2345.084  mm,	Y =   -99.346  mm,	Z =   921.026  mm,
	W =   -40.224 deg,	P =    17.491 deg,	R =   -11.143 deg
   GP2:
	UF : 0, UT : 1,
	J1=    90.000 deg,	J2=    90.000 deg
};
P[913]{
   GP1:
	UF : 1, UT : 1,		CONFIG : 'N U T, 0, 0, 0',
	X =  2345.241  mm,	Y =  -143.403  mm,	Z =   870.965  mm,
	W =   -36.126 deg,	P =    18.220 deg,	R =    -8.746 deg
   GP2:
	UF : 0, UT : 1,
	J1=    89.999 deg,	J2=    90.000 deg
};
P[914]{
   GP1:
	UF : 1, UT : 1,		CONFIG : 'N U T, 0, 0, 0',
	X =  2282.648  mm,	Y =  -109.823  mm,	Z =   871.166  mm,
	W =   -36.146 deg,	P =    18.219 deg,	R =    -8.768 deg
   GP2:
	UF : 0, UT : 1,
	J1=    90.000 deg,	J2=    90.000 deg
};
P[915]{
   GP1:
	UF : 1, UT : 1,		CONFIG : 'N U T, 0, 0, 0',
	X =  2345.084  mm,	Y =   -99.346  mm,	Z =  1021.026  mm,
	W =   -40.224 deg,	P =    17.491 deg,	R =   -11.143 deg
   GP2:
	UF : 0, UT : 1,
	J1=    90.000 deg,	J2=    90.000 deg
};
P[916]{
   GP1:
	UF : 1, UT : 1,		CONFIG : 'N U T, 0, 0, 0',
	X =  2403.931  mm,	Y =  -153.062  mm,	Z =   942.017  mm,
	W =   -14.995 deg,	P =    37.514 deg,	R =   -38.639 deg
   GP2:
	UF : 0, UT : 1,
	J1=    90.000 deg,	J2=    90.000 deg
};
P[917]{
   GP1:
	UF : 1, UT : 1,		CONFIG : 'N U T, 0, 0, 0',
	X =  2347.931  mm,	Y =  -146.592  mm,	Z =   870.891  mm,
	W =   -14.995 deg,	P =    37.514 deg,	R =   -38.639 deg
   GP2:
	UF : 0, UT : 1,
	J1=    90.000 deg,	J2=    90.000 deg
};
P[918]{
   GP1:
	UF : 1, UT : 1,		CONFIG : 'N U T, 0, 0, 0',
	X =  2337.717  mm,	Y =  -167.449  mm,	Z =   870.891  mm,
	W =   -14.995 deg,	P =    37.514 deg,	R =   -38.639 deg
   GP2:
	UF : 0, UT : 1,
	J1=    90.000 deg,	J2=    90.000 deg
};
P[919]{
   GP1:
	UF : 1, UT : 1,		CONFIG : 'N U T, 0, 0, 0',
	X =  2375.358  mm,	Y =  -188.860  mm,	Z =   936.517  mm,
	W =   -11.991 deg,	P =    31.145 deg,	R =   -43.623 deg
   GP2:
	UF : 0, UT : 1,
	J1=    90.000 deg,	J2=    90.000 deg
};
P[920]{
   GP1:
	UF : 1, UT : 1,		CONFIG : 'N U T, 0, 0, 0',
	X =  2241.084  mm,	Y =  -176.345  mm,	Z =  1066.026  mm,
	W =    39.867 deg,	P =   -18.417 deg,	R =   -24.499 deg
   GP2:
	UF : 0, UT : 1,
	J1=    90.000 deg,	J2=    90.000 deg
};
P[921]{
   GP1:
	UF : 1, UT : 1,		CONFIG : 'N U T, 0, 0, 0',
	X =  2267.739  mm,	Y =  -132.899  mm,	Z =   875.644  mm,
	W =    39.860 deg,	P =   -18.420 deg,	R =   -24.496 deg
   GP2:
	UF : 0, UT : 1,
	J1=    90.000 deg,	J2=    90.000 deg
};
P[922]{
   GP1:
	UF : 1, UT : 1,		CONFIG : 'N U T, 0, 0, 0',
	X =  2334.568  mm,	Y =  -169.227  mm,	Z =   875.761  mm,
	W =    34.466 deg,	P =   -19.855 deg,	R =   -14.827 deg
   GP2:
	UF : 0, UT : 1,
	J1=    90.000 deg,	J2=    90.000 deg
};
P[923]{
   GP1:
	UF : 1, UT : 1,		CONFIG : 'N U T, 0, 0, 0',
	X =  2241.084  mm,	Y =  -176.345  mm,	Z =  1066.025  mm,
	W =    39.866 deg,	P =   -18.417 deg,	R =   -39.014 deg
   GP2:
	UF : 0, UT : 1,
	J1=    90.000 deg,	J2=    90.000 deg
};
P[924]{
   GP1:
	UF : 1, UT : 1,		CONFIG : 'N U T, 0, 0, 0',
	X =  1615.083  mm,	Y =   143.655  mm,	Z =  1238.025  mm,
	W =    39.866 deg,	P =   -18.417 deg,	R =   -39.014 deg
   GP2:
	UF : 0, UT : 1,
	J1=    90.000 deg,	J2=    90.000 deg
};
P[925]{
   GP1:
	UF : 1, UT : 1,		CONFIG : 'N U T, 0, 0, 0',
	X =  1426.736  mm,	Y =   -88.930  mm,	Z =  1060.273  mm,
	W =    35.942 deg,	P =   -29.145 deg,	R =   -48.109 deg
   GP2:
	UF : 0, UT : 1,
	J1=    90.000 deg,	J2=    90.000 deg
};
P[926]{
   GP1:
	UF : 1, UT : 1,		CONFIG : 'N U T, 0, 0, 0',
	X =  1598.736  mm,	Y =   -66.432  mm,	Z =   872.868  mm,
	W =    35.824 deg,	P =   -29.280 deg,	R =   -48.048 deg
   GP2:
	UF : 0, UT : 1,
	J1=    89.999 deg,	J2=    90.000 deg
};
P[927]{
   GP1:
	UF : 1, UT : 1,		CONFIG : 'N U T, 0, 0, 0',
	X =  1652.530  mm,	Y =  -479.384  mm,	Z =   873.834  mm,
	W =    44.626 deg,	P =    -6.633 deg,	R =   -75.290 deg
   GP2:
	UF : 0, UT : 1,
	J1=    89.999 deg,	J2=    90.000 deg
};
P[928]{
   GP1:
	UF : 1, UT : 1,		CONFIG : 'N U T, 0, 0, 0',
	X =  1441.417  mm,	Y =  -441.770  mm,	Z =  1074.656  mm,
	W =    48.178 deg,	P =   -19.898 deg,	R =   -92.005 deg
   GP2:
	UF : 0, UT : 1,
	J1=    90.000 deg,	J2=    90.000 deg
};
P[929]{
   GP1:
	UF : 1, UT : 1,		CONFIG : 'N U T, 0, 0, -1',
	X =  1441.417  mm,	Y =  -118.913  mm,	Z =  1074.656  mm,
	W =    -2.520 deg,	P =    51.125 deg,	R =   157.822 deg
   GP2:
	UF : 0, UT : 1,
	J1=    90.000 deg,	J2=    90.000 deg
};
P[930]{
   GP1:
	UF : 1, UT : 1,		CONFIG : 'N U T, 0, 0, 0',
	X =  1685.416  mm,	Y =   -62.913  mm,	Z =  1074.656  mm,
	W =    -3.706 deg,	P =    39.360 deg,	R =     3.645 deg
   GP2:
	UF : 0, UT : 1,
	J1=    90.000 deg,	J2=    90.000 deg
};
P[931]{
   GP1:
	UF : 1, UT : 1,		CONFIG : 'N U T, 0, 0, 0',
	X =  1611.253  mm,	Y =   -63.766  mm,	Z =   866.535  mm,
	W =    -3.351 deg,	P =    44.836 deg,	R =     3.194 deg
   GP2:
	UF : 0, UT : 1,
	J1=    89.995 deg,	J2=    90.000 deg
};
P[932]{
   GP1:
	UF : 1, UT : 1,		CONFIG : 'N U T, 0, 0, 0',
	X =  1668.640  mm,	Y =  -484.243  mm,	Z =   867.735  mm,
	W =   -41.394 deg,	P =    19.465 deg,	R =   -61.379 deg
   GP2:
	UF : 0, UT : 1,
	J1=    90.000 deg,	J2=    90.000 deg
};
P[933]{
   GP1:
	UF : 1, UT : 1,		CONFIG : 'N U T, 0, 0, 0',
	X =  1815.595  mm,	Y =  -400.803  mm,	Z =  1004.765  mm,
	W =   -43.547 deg,	P =    12.687 deg,	R =   -45.705 deg
   GP2:
	UF : 0, UT : 1,
	J1=    90.000 deg,	J2=    90.000 deg
};
P[934]{
   GP1:
	UF : 1, UT : 1,		CONFIG : 'N U T, 0, 0, 0',
	X =  1833.172  mm,	Y =   137.472  mm,	Z =  1065.903  mm,
	W =    -8.569 deg,	P =    33.778 deg,	R =   -31.530 deg
   GP2:
	UF : 0, UT : 1,
	J1=    90.000 deg,	J2=    90.000 deg
};
P[935]{
   GP1:
	UF : 1, UT : 1,		CONFIG : 'N U T, 0, 0, 0',
	X =   730.446  mm,	Y =   700.194  mm,	Z =  1357.060  mm,
	W =    -8.561 deg,	P =    33.775 deg,	R =    -6.417 deg
   GP2:
	UF : 0, UT : 1,
	J1=    90.000 deg,	J2=    90.000 deg
};
P[936]{
   GP1:
	UF : 1, UT : 1,		CONFIG : 'N U T, 0, 0, 0',
	X =  2460.862  mm,	Y =  1574.474  mm,	Z =  1293.677  mm,
	W =    34.631 deg,	P =   -20.439 deg,	R =   -45.641 deg
   GP2:
	UF : 0, UT : 1,
	J1=    90.000 deg,	J2=    80.000 deg
};
P[937]{
   GP1:
	UF : 1, UT : 1,		CONFIG : 'N U T, 0, 0, 0',
	X =  2554.185  mm,	Y =  1608.224  mm,	Z =   812.612  mm,
	W =    36.017 deg,	P =   -29.586 deg,	R =   -62.799 deg
   GP2:
	UF : 0, UT : 1,
	J1=    90.000 deg,	J2=    80.000 deg
};
P[938]{
   GP1:
	UF : 1, UT : 1,		CONFIG : 'N U T, 0, 0, 0',
	X =  2770.210  mm,	Y =  1515.223  mm,	Z =   663.612  mm,
	W =    36.017 deg,	P =   -29.586 deg,	R =   -64.860 deg
   GP2:
	UF : 0, UT : 1,
	J1=    90.000 deg,	J2=    80.000 deg
};
P[939]{
   GP1:
	UF : 1, UT : 1,		CONFIG : 'N U T, 0, 0, 0',
	X =  2859.251  mm,	Y =  1470.161  mm,	Z =   622.793  mm,
	W =    21.035 deg,	P =   -48.595 deg,	R =   -52.950 deg
   GP2:
	UF : 0, UT : 1,
	J1=    89.999 deg,	J2=    80.000 deg
};
P[940]{
   GP1:
	UF : 1, UT : 1,		CONFIG : 'N U T, 0, 0, 0',
	X =  2862.590  mm,	Y =  1519.336  mm,	Z =   614.634  mm,
	W =    25.659 deg,	P =   -39.366 deg,	R =   -46.936 deg
   GP2:
	UF : 0, UT : 1,
	J1=    89.999 deg,	J2=    80.000 deg
};
P[941]{
   GP1:
	UF : 1, UT : 1,		CONFIG : 'N U T, 0, 0, 0',
	X =  2848.858  mm,	Y =  1554.917  mm,	Z =   605.833  mm,
	W =    38.517 deg,	P =   -13.826 deg,	R =   -52.000 deg
   GP2:
	UF : 0, UT : 1,
	J1=    89.999 deg,	J2=    80.000 deg
};
P[942]{
   GP1:
	UF : 1, UT : 1,		CONFIG : 'N U T, 0, 0, 0',
	X =  2816.955  mm,	Y =  1578.946  mm,	Z =   600.178  mm,
	W =    36.558 deg,	P =     2.413 deg,	R =   -39.556 deg
   GP2:
	UF : 0, UT : 1,
	J1=    90.000 deg,	J2=    80.000 deg
};
P[943]{
   GP1:
	UF : 1, UT : 1,		CONFIG : 'N U T, 0, 0, 0',
	X =  2767.863  mm,	Y =  1609.158  mm,	Z =   594.729  mm,
	W =    36.709 deg,	P =    -5.347 deg,	R =   -45.355 deg
   GP2:
	UF : 0, UT : 1,
	J1=    90.000 deg,	J2=    80.000 deg
};
P[944]{
   GP1:
	UF : 1, UT : 1,		CONFIG : 'N U T, 0, 0, 0',
	X =  2666.921  mm,	Y =  1574.106  mm,	Z =   705.413  mm,
	W =    36.699 deg,	P =    -5.422 deg,	R =   -45.347 deg
   GP2:
	UF : 0, UT : 1,
	J1=    90.000 deg,	J2=    80.000 deg
};
P[945]{
   GP1:
	UF : 1, UT : 1,		CONFIG : 'N U T, 0, 0, 0',
	X =  2623.443  mm,	Y =  1700.524  mm,	Z =   713.976  mm,
	W =   -50.219 deg,	P =    -7.077 deg,	R =    46.580 deg
   GP2:
	UF : 0, UT : 1,
	J1=    90.000 deg,	J2=    80.000 deg
};
P[946]{
   GP1:
	UF : 1, UT : 1,		CONFIG : 'N U T, 0, 0, 0',
	X =  2764.713  mm,	Y =  1617.218  mm,	Z =   592.857  mm,
	W =   -50.556 deg,	P =     -.080 deg,	R =    52.376 deg
   GP2:
	UF : 0, UT : 1,
	J1=    89.999 deg,	J2=    80.000 deg
};
P[947]{
   GP1:
	UF : 1, UT : 1,		CONFIG : 'N U T, 0, 0, 0',
	X =  2778.189  mm,	Y =  1640.751  mm,	Z =   588.691  mm,
	W =   -50.492 deg,	P =     -.105 deg,	R =    52.361 deg
   GP2:
	UF : 0, UT : 1,
	J1=    89.999 deg,	J2=    80.000 deg
};
P[948]{
   GP1:
	UF : 1, UT : 1,		CONFIG : 'N U T, 0, 0, 0',
	X =  2619.398  mm,	Y =  1698.477  mm,	Z =   698.692  mm,
	W =   -54.549 deg,	P =   -20.575 deg,	R =    64.434 deg
   GP2:
	UF : 0, UT : 1,
	J1=    90.000 deg,	J2=    80.000 deg
};
P[949]{
   GP1:
	UF : 1, UT : 1,		CONFIG : 'N U T, 0, 0, 0',
	X =  1431.673  mm,	Y =   731.089  mm,	Z =  1754.089  mm,
	W =    28.012 deg,	P =   -23.444 deg,	R =   -34.782 deg
   GP2:
	UF : 0, UT : 1,
	J1=    90.000 deg,	J2=    80.000 deg
};
P[950]{
   GP1:
	UF : 1, UT : 1,		CONFIG : 'N U B, 0, 0, 0',
	X =   390.614  mm,	Y =     -.024  mm,	Z =  2434.016  mm,
	W =     -.021 deg,	P =   -39.773 deg,	R =      .020 deg
   GP2:
	UF : 0, UT : 1,
	J1=    90.000 deg,	J2=    80.000 deg
};
P[951]{
   GP1:
	UF : 1, UT : 1,
	J1=   -67.228 deg,	J2=   -42.143 deg,	J3=    26.623 deg,
	J4=   -68.823 deg,	J5=  -105.727 deg,	J6=   144.671 deg
   GP2:
	UF : 0, UT : 1,
	J1=   -90.000 deg,	J2=    90.000 deg
};
P[952]{
   GP1:
	UF : 1, UT : 1,		CONFIG : 'N U T, 0, 0, 0',
	X =   921.742  mm,	Y =  -602.772  mm,	Z =  1080.858  mm,
	W =   -52.537 deg,	P =    -3.928 deg,	R =    83.324 deg
   GP2:
	UF : 0, UT : 1,
	J1=   -90.000 deg,	J2=    90.000 deg
};
P[953]{
   GP1:
	UF : 1, UT : 1,		CONFIG : 'N U T, 0, 0, 0',
	X =  1662.139  mm,	Y =  -563.740  mm,	Z =   954.127  mm,
	W =   -52.527 deg,	P =    -3.934 deg,	R =    60.639 deg
   GP2:
	UF : 0, UT : 1,
	J1=   -90.000 deg,	J2=    90.000 deg
};
P[954]{
   GP1:
	UF : 1, UT : 1,		CONFIG : 'N U T, 0, 0, 0',
	X =  1699.178  mm,	Y =  -604.727  mm,	Z =   864.903  mm,
	W =   -44.004 deg,	P =    -1.784 deg,	R =    59.349 deg
   GP2:
	UF : 0, UT : 1,
	J1=   -90.000 deg,	J2=    90.000 deg
};
P[955]{
   GP1:
	UF : 1, UT : 1,		CONFIG : 'N U T, 0, 0, 0',
	X =  1939.327  mm,	Y =  -157.054  mm,	Z =   862.507  mm,
	W =   -44.919 deg,	P =    -3.099 deg,	R =    71.282 deg
   GP2:
	UF : 0, UT : 1,
	J1=   -90.000 deg,	J2=    90.000 deg
};
P[956]{
   GP1:
	UF : 1, UT : 1,		CONFIG : 'N U T, 0, 0, 0',
	X =  1947.551  mm,	Y =  -143.847  mm,	Z =   939.637  mm,
	W =   -64.247 deg,	P =    -5.308 deg,	R =    92.033 deg
   GP2:
	UF : 0, UT : 1,
	J1=   -90.000 deg,	J2=    90.000 deg
};
P[957]{
   GP1:
	UF : 1, UT : 1,		CONFIG : 'N U T, 0, 0, 0',
	X =  1339.858  mm,	Y =  -518.344  mm,	Z =   958.778  mm,
	W =   -68.704 deg,	P =    -3.326 deg,	R =    72.634 deg
   GP2:
	UF : 0, UT : 1,
	J1=   -90.000 deg,	J2=    90.000 deg
};
P[958]{
   GP1:
	UF : 1, UT : 1,		CONFIG : 'N U T, 0, 0, 0',
	X =  1178.463  mm,	Y =  -576.131  mm,	Z =   850.740  mm,
	W =     5.796 deg,	P =    -2.160 deg,	R =   -21.237 deg
   GP2:
	UF : 0, UT : 1,
	J1=   -90.000 deg,	J2=    90.000 deg
};
P[959]{
   GP1:
	UF : 1, UT : 1,		CONFIG : 'N U T, 0, 0, 0',
	X =  1259.408  mm,	Y =  -666.652  mm,	Z =   959.172  mm,
	W =    58.410 deg,	P =     1.273 deg,	R =   -88.963 deg
   GP2:
	UF : 0, UT : 1,
	J1=   -90.000 deg,	J2=    90.000 deg
};
P[960]{
   GP1:
	UF : 1, UT : 1,		CONFIG : 'N U T, 0, 0, 0',
	X =  1642.096  mm,	Y =  -668.648  mm,	Z =   941.442  mm,
	W =    46.641 deg,	P =   -16.556 deg,	R =   -73.967 deg
   GP2:
	UF : 0, UT : 1,
	J1=   -90.000 deg,	J2=    90.000 deg
};
P[961]{
   GP1:
	UF : 1, UT : 1,		CONFIG : 'N U T, 0, 0, 0',
	X =  1680.196  mm,	Y =  -661.782  mm,	Z =   867.291  mm,
	W =    44.399 deg,	P =   -17.018 deg,	R =   -72.718 deg
   GP2:
	UF : 0, UT : 1,
	J1=   -90.000 deg,	J2=    90.000 deg
};
P[962]{
   GP1:
	UF : 1, UT : 1,		CONFIG : 'N U T, 0, 0, 0',
	X =  1679.681  mm,	Y =  -677.294  mm,	Z =   868.712  mm,
	W =    44.369 deg,	P =   -17.049 deg,	R =   -59.242 deg
   GP2:
	UF : 0, UT : 1,
	J1=   -90.000 deg,	J2=    90.000 deg
};
P[963]{
   GP1:
	UF : 1, UT : 1,		CONFIG : 'N U T, 0, 0, 0',
	X =  1689.612  mm,	Y =  -701.782  mm,	Z =   867.996  mm,
	W =    44.379 deg,	P =   -17.045 deg,	R =   -47.908 deg
   GP2:
	UF : 0, UT : 1,
	J1=   -90.000 deg,	J2=    90.000 deg
};
P[964]{
   GP1:
	UF : 1, UT : 1,		CONFIG : 'N U T, 0, 0, 0',
	X =  1888.332  mm,	Y = -1073.282  mm,	Z =   870.872  mm,
	W =    44.370 deg,	P =   -17.046 deg,	R =   -47.907 deg
   GP2:
	UF : 0, UT : 1,
	J1=   -90.000 deg,	J2=    90.000 deg
};
P[965]{
   GP1:
	UF : 1, UT : 1,		CONFIG : 'N U T, 0, 0, 0',
	X =  1720.695  mm,	Y =  -903.847  mm,	Z =   939.638  mm,
	W =    45.135 deg,	P =   -18.028 deg,	R =   -72.006 deg
   GP2:
	UF : 0, UT : 1,
	J1=   -90.000 deg,	J2=    90.000 deg
};
P[966]{
   GP1:
	UF : 1, UT : 1,		CONFIG : 'N U T, 0, 0, 0',
	X =  1150.537  mm,	Y =  -903.847  mm,	Z =   939.637  mm,
	W =    45.135 deg,	P =   -18.028 deg,	R =   -72.006 deg
   GP2:
	UF : 0, UT : 1,
	J1=   -90.000 deg,	J2=    90.000 deg
};
P[967]{
   GP1:
	UF : 1, UT : 1,		CONFIG : 'N U B, 0, 0, 0',
	X =   390.614  mm,	Y =     -.024  mm,	Z =  2434.015  mm,
	W =     -.021 deg,	P =   -39.773 deg,	R =      .020 deg
   GP2:
	UF : 0, UT : 1,
	J1=   -90.000 deg,	J2=    90.000 deg
};
P[968]{
   GP1:
	UF : 1, UT : 1,
	J1=    31.349 deg,	J2=   -58.835 deg,	J3=    14.453 deg,
	J4=   -25.392 deg,	J5=   -40.935 deg,	J6=    86.768 deg
   GP2:
	UF : 0, UT : 1,
	J1=   -90.000 deg,	J2=   -90.000 deg
};
P[969]{
   GP1:
	UF : 1, UT : 1,		CONFIG : 'N U T, 0, 0, 0',
	X =  1658.982  mm,	Y =   679.545  mm,	Z =   922.923  mm,
	W =   -53.210 deg,	P =    -2.950 deg,	R =    86.737 deg
   GP2:
	UF : 0, UT : 1,
	J1=   -90.000 deg,	J2=   -90.000 deg
};
P[970]{
   GP1:
	UF : 1, UT : 1,		CONFIG : 'N U T, 0, 0, 0',
	X =  1676.975  mm,	Y =   666.399  mm,	Z =   865.172  mm,
	W =   -44.636 deg,	P =    -2.340 deg,	R =    86.168 deg
   GP2:
	UF : 0, UT : 1,
	J1=   -90.000 deg,	J2=   -90.000 deg
};
P[971]{
   GP1:
	UF : 1, UT : 1,		CONFIG : 'N U T, 0, 0, 0',
	X =  1679.488  mm,	Y =   683.862  mm,	Z =   864.814  mm,
	W =   -44.615 deg,	P =    -2.365 deg,	R =    73.000 deg
   GP2:
	UF : 0, UT : 1,
	J1=   -90.000 deg,	J2=   -90.000 deg
};
P[972]{
   GP1:
	UF : 1, UT : 1,		CONFIG : 'N U T, 0, 0, 0',
	X =  1688.681  mm,	Y =   703.537  mm,	Z =   862.970  mm,
	W =   -44.588 deg,	P =    -2.365 deg,	R =    57.125 deg
   GP2:
	UF : 0, UT : 1,
	J1=   -90.000 deg,	J2=   -90.000 deg
};
P[973]{
   GP1:
	UF : 1, UT : 1,		CONFIG : 'N U T, 0, 0, 0',
	X =  1890.870  mm,	Y =  1078.356  mm,	Z =   862.379  mm,
	W =   -43.116 deg,	P =   -12.585 deg,	R =    51.673 deg
   GP2:
	UF : 0, UT : 1,
	J1=   -90.000 deg,	J2=   -90.000 deg
};
P[974]{
   GP1:
	UF : 1, UT : 1,		CONFIG : 'N U T, 0, 0, 0',
	X =  1751.245  mm,	Y =  1086.047  mm,	Z =   952.940  mm,
	W =   -46.336 deg,	P =   -33.058 deg,	R =    48.624 deg
   GP2:
	UF : 0, UT : 1,
	J1=   -90.000 deg,	J2=   -90.000 deg
};
P[975]{
   GP1:
	UF : 1, UT : 1,		CONFIG : 'N U T, 0, 0, 0',
	X =  1119.126  mm,	Y =  1086.046  mm,	Z =   952.940  mm,
	W =   -46.336 deg,	P =   -33.058 deg,	R =    48.624 deg
   GP2:
	UF : 0, UT : 1,
	J1=   -90.000 deg,	J2=   -90.000 deg
};
P[976]{
   GP1:
	UF : 1, UT : 1,		CONFIG : 'N U B, 0, 0, 0',
	X =   390.614  mm,	Y =     -.024  mm,	Z =  2434.016  mm,
	W =     -.021 deg,	P =   -39.773 deg,	R =      .020 deg
   GP2:
	UF : 0, UT : 1,
	J1=   -90.000 deg,	J2=   -90.000 deg
};
P[977]{
   GP1:
	UF : 1, UT : 1,		CONFIG : 'N U T, 0, 0, 0',
	X =  1013.045  mm,	Y =  -777.257  mm,	Z =  1208.287  mm,
	W =    -1.627 deg,	P =    35.013 deg,	R =    16.289 deg
   GP2:
	UF : 0, UT : 1,
	J1=    90.000 deg,	J2=   -90.000 deg
};
P[978]{
   GP1:
	UF : 1, UT : 1,		CONFIG : 'N U T, 0, 0, 0',
	X =  1891.794  mm,	Y =  -123.744  mm,	Z =    89.423  mm,
	W =   -43.304 deg,	P =     8.281 deg,	R =    89.437 deg
   GP2:
	UF : 0, UT : 1,
	J1=    90.000 deg,	J2=   -90.000 deg
};
P[979]{
   GP1:
	UF : 1, UT : 1,		CONFIG : 'N U T, 0, 0, 0',
	X =  1964.710  mm,	Y =   -77.630  mm,	Z =    75.842  mm,
	W =   -43.304 deg,	P =     8.281 deg,	R =    95.107 deg
   GP2:
	UF : 0, UT : 1,
	J1=    90.000 deg,	J2=   -90.000 deg
};
P[980]{
   GP1:
	UF : 1, UT : 1,		CONFIG : 'N U T, 0, 0, 0',
	X =  2022.737  mm,	Y =   -48.948  mm,	Z =   -36.034  mm,
	W =   -39.351 deg,	P =    23.856 deg,	R =   118.022 deg
   GP2:
	UF : 0, UT : 1,
	J1=    90.000 deg,	J2=   -90.000 deg
};
P[981]{
   GP1:
	UF : 1, UT : 1,		CONFIG : 'N U T, 0, 0, 1',
	X =  2042.531  mm,	Y =   -19.520  mm,	Z =   -34.591  mm,
	W =   -39.343 deg,	P =    23.911 deg,	R =   138.810 deg
   GP2:
	UF : 0, UT : 1,
	J1=    89.998 deg,	J2=   -90.000 deg
};
P[982]{
   GP1:
	UF : 1, UT : 1,		CONFIG : 'N U T, 0, 0, 0',
	X =  1966.026  mm,	Y =   -53.845  mm,	Z =   115.121  mm,
	W =   -43.304 deg,	P =     8.281 deg,	R =   116.653 deg
   GP2:
	UF : 0, UT : 1,
	J1=    90.000 deg,	J2=   -90.000 deg
};
P[983]{
   GP1:
	UF : 1, UT : 1,		CONFIG : 'N U T, 0, 0, 0',
	X =  1707.026  mm,	Y =  -401.845  mm,	Z =   180.120  mm,
	W =   -43.304 deg,	P =     8.281 deg,	R =   116.653 deg
   GP2:
	UF : 0, UT : 1,
	J1=    90.000 deg,	J2=   -90.000 deg
};
P[984]{
   GP1:
	UF : 1, UT : 1,		CONFIG : 'N U T, 0, 0, 0',
	X =  1624.711  mm,	Y = -1090.629  mm,	Z =   272.128  mm,
	W =    43.884 deg,	P =    -2.387 deg,	R =     2.487 deg
   GP2:
	UF : 0, UT : 1,
	J1=    90.000 deg,	J2=   -90.000 deg
};
P[985]{
   GP1:
	UF : 1, UT : 1,		CONFIG : 'N U T, 0, 0, 0',
	X =  2631.710  mm,	Y =  -986.630  mm,	Z =    81.842  mm,
	W =    43.884 deg,	P =    -2.387 deg,	R =     2.487 deg
   GP2:
	UF : 0, UT : 1,
	J1=    90.000 deg,	J2=   -90.000 deg
};
P[986]{
   GP1:
	UF : 1, UT : 1,		CONFIG : 'N U T, 0, 0, 0',
	X =  2642.691  mm,	Y =  -923.695  mm,	Z =   -21.197  mm,
	W =    44.909 deg,	P =    -2.402 deg,	R =     2.450 deg
   GP2:
	UF : 0, UT : 1,
	J1=    90.000 deg,	J2=   -90.000 deg
};
P[987]{
   GP1:
	UF : 1, UT : 1,		CONFIG : 'N U T, 0, 0, 0',
	X =  2675.893  mm,	Y =  -923.999  mm,	Z =   -21.545  mm,
	W =    44.951 deg,	P =    -2.429 deg,	R =     2.434 deg
   GP2:
	UF : 0, UT : 1,
	J1=    90.000 deg,	J2=   -90.000 deg
};
P[988]{
   GP1:
	UF : 1, UT : 1,		CONFIG : 'N U T, 0, 0, 0',
	X =  2687.713  mm,	Y =  -922.067  mm,	Z =   -21.309  mm,
	W =    43.920 deg,	P =    11.009 deg,	R =     5.127 deg
   GP2:
	UF : 0, UT : 1,
	J1=    90.000 deg,	J2=   -90.000 deg
};
P[989]{
   GP1:
	UF : 1, UT : 1,		CONFIG : 'N U T, 0, 0, 0',
	X =  2700.218  mm,	Y =  -906.405  mm,	Z =   -18.902  mm,
	W =    43.903 deg,	P =    11.008 deg,	R =     2.411 deg
   GP2:
	UF : 0, UT : 1,
	J1=    90.000 deg,	J2=   -90.000 deg
};
P[990]{
   GP1:
	UF : 1, UT : 1,		CONFIG : 'N U T, 0, 0, 0',
	X =  2687.411  mm,	Y =  -983.390  mm,	Z =    66.919  mm,
	W =    43.915 deg,	P =    11.001 deg,	R =   -22.994 deg
   GP2:
	UF : 0, UT : 1,
	J1=    90.000 deg,	J2=   -90.000 deg
};
P[991]{
   GP1:
	UF : 1, UT : 1,		CONFIG : 'N U T, 0, 0, 0',
	X =  1931.038  mm,	Y = -1008.724  mm,	Z =   170.682  mm,
	W =    44.948 deg,	P =    -2.436 deg,	R =    -7.767 deg
   GP2:
	UF : 0, UT : 1,
	J1=    90.000 deg,	J2=   -90.000 deg
};
P[992]{
   GP1:
	UF : 1, UT : 1,		CONFIG : 'N U T, 0, 0, 0',
	X =  1931.038  mm,	Y = -1008.725  mm,	Z =   253.683  mm,
	W =   -41.218 deg,	P =   -19.941 deg,	R =   -32.390 deg
   GP2:
	UF : 0, UT : 1,
	J1=    90.000 deg,	J2=   -90.000 deg
};
P[993]{
   GP1:
	UF : 1, UT : 1,		CONFIG : 'N U T, 0, 0, 0',
	X =  2543.038  mm,	Y =  -803.725  mm,	Z =   184.397  mm,
	W =   -38.746 deg,	P =   -26.390 deg,	R =   -19.221 deg
   GP2:
	UF : 0, UT : 1,
	J1=    90.000 deg,	J2=   -90.000 deg
};
P[994]{
   GP1:
	UF : 1, UT : 1,		CONFIG : 'N U T, 0, 0, 0',
	X =  2602.037  mm,	Y =  -803.725  mm,	Z =    84.396  mm,
	W =   -43.420 deg,	P =   -13.149 deg,	R =   -17.628 deg
   GP2:
	UF : 0, UT : 1,
	J1=    90.000 deg,	J2=   -90.000 deg
};
P[995]{
   GP1:
	UF : 1, UT : 1,		CONFIG : 'N U T, 0, 0, 0',
	X =  2646.853  mm,	Y =  -840.409  mm,	Z =   -23.316  mm,
	W =   -40.207 deg,	P =    -8.263 deg,	R =    -9.650 deg
   GP2:
	UF : 0, UT : 1,
	J1=    90.000 deg,	J2=   -90.000 deg
};
P[996]{
   GP1:
	UF : 1, UT : 1,		CONFIG : 'N U T, 0, 0, 0',
	X =  2673.374  mm,	Y =  -841.195  mm,	Z =   -24.120  mm,
	W =   -44.987 deg,	P =    -1.268 deg,	R =    -1.270 deg
   GP2:
	UF : 0, UT : 1,
	J1=    90.000 deg,	J2=   -90.000 deg
};
P[997]{
   GP1:
	UF : 1, UT : 1,		CONFIG : 'N U T, 0, 0, 0',
	X =  2692.519  mm,	Y =  -849.008  mm,	Z =   -26.521  mm,
	W =   -44.971 deg,	P =     1.298 deg,	R =   -25.927 deg
   GP2:
	UF : 0, UT : 1,
	J1=    89.999 deg,	J2=   -90.000 deg
};
P[998]{
   GP1:
	UF : 1, UT : 1,		CONFIG : 'N U T, 0, 0, 0',
	X =  2702.206  mm,	Y =  -866.851  mm,	Z =   -24.735  mm,
	W =   -44.924 deg,	P =    -1.260 deg,	R =   -28.515 deg
   GP2:
	UF : 0, UT : 1,
	J1=    90.000 deg,	J2=   -90.000 deg
};
P[999]{
   GP1:
	UF : 1, UT : 1,		CONFIG : 'N U T, 0, 0, 0',
	X =  2602.037  mm,	Y =  -803.725  mm,	Z =    84.396  mm,
	W =   -43.420 deg,	P =   -13.149 deg,	R =   -17.628 deg
   GP2:
	UF : 0, UT : 1,
	J1=    90.000 deg,	J2=   -90.000 deg
};
P[1000]{
   GP1:
	UF : 1, UT : 1,		CONFIG : 'N U T, 0, 0, 0',
	X =  2543.038  mm,	Y =  -803.725  mm,	Z =   184.397  mm,
	W =   -36.633 deg,	P =   -31.550 deg,	R =   -20.246 deg
   GP2:
	UF : 0, UT : 1,
	J1=    90.000 deg,	J2=   -90.000 deg
};
P[1001]{
   GP1:
	UF : 1, UT : 1,		CONFIG : 'N U T, 0, 0, 0',
	X =  1631.038  mm,	Y = -1008.725  mm,	Z =   203.683  mm,
	W =   -41.218 deg,	P =   -19.941 deg,	R =   -32.390 deg
   GP2:
	UF : 0, UT : 1,
	J1=    90.000 deg,	J2=   -90.000 deg
};
P[1002]{
   GP1:
	UF : 1, UT : 1,		CONFIG : 'N U T, 0, 0, 0',
	X =  1624.710  mm,	Y =  -283.630  mm,	Z =   237.842  mm,
	W =    43.884 deg,	P =    -2.387 deg,	R =     2.487 deg
   GP2:
	UF : 0, UT : 1,
	J1=    90.000 deg,	J2=   -90.000 deg
};
P[1003]{
   GP1:
	UF : 1, UT : 1,		CONFIG : 'N U T, 0, 0, 0',
	X =  1594.691  mm,	Y =  -106.040  mm,	Z =    30.842  mm,
	W =    43.884 deg,	P =    -2.387 deg,	R =     2.487 deg
   GP2:
	UF : 0, UT : 1,
	J1=    90.000 deg,	J2=   -90.000 deg
};
P[1004]{
   GP1:
	UF : 1, UT : 1,		CONFIG : 'N U T, 0, 0, 0',
	X =  1590.451  mm,	Y =   -18.944  mm,	Z =   -34.547  mm,
	W =    39.221 deg,	P =   -24.029 deg,	R =    26.552 deg
   GP2:
	UF : 0, UT : 1,
	J1=    90.000 deg,	J2=   -90.000 deg
};
P[1005]{
   GP1:
	UF : 1, UT : 1,		CONFIG : 'N U T, 0, 0, 0',
	X =  1578.966  mm,	Y =   -21.965  mm,	Z =   -37.747  mm,
	W =    43.587 deg,	P =   -12.502 deg,	R =    37.180 deg
   GP2:
	UF : 0, UT : 1,
	J1=    90.000 deg,	J2=   -90.000 deg
};
P[1006]{
   GP1:
	UF : 1, UT : 1,		CONFIG : 'N U T, 0, 0, 0',
	X =  1573.690  mm,	Y =   -24.800  mm,	Z =   -40.057  mm,
	W =    44.958 deg,	P =    -2.233 deg,	R =    47.234 deg
   GP2:
	UF : 0, UT : 1,
	J1=    90.000 deg,	J2=   -90.000 deg
};
P[1007]{
   GP1:
	UF : 1, UT : 1,		CONFIG : 'N U T, 0, 0, 0',
	X =  1543.842  mm,	Y =   -53.176  mm,	Z =   -39.928  mm,
	W =    44.961 deg,	P =    -2.235 deg,	R =    47.243 deg
   GP2:
	UF : 0, UT : 1,
	J1=    90.000 deg,	J2=   -90.000 deg
};
P[1008]{
   GP1:
	UF : 1, UT : 1,		CONFIG : 'N U T, 0, 0, 0',
	X =  1527.813  mm,	Y =   -57.039  mm,	Z =   -38.383  mm,
	W =    34.021 deg,	P =   -31.373 deg,	R =    36.125 deg
   GP2:
	UF : 0, UT : 1,
	J1=    90.000 deg,	J2=   -90.000 deg
};
P[1009]{
   GP1:
	UF : 1, UT : 1,		CONFIG : 'N U T, 0, 0, 0',
	X =  1513.122  mm,	Y =   -42.298  mm,	Z =   -40.119  mm,
	W =   -41.192 deg,	P =   -19.991 deg,	R =    73.659 deg
   GP2:
	UF : 0, UT : 1,
	J1=    90.000 deg,	J2=   -90.000 deg
};
P[1010]{
   GP1:
	UF : 1, UT : 1,		CONFIG : 'N U T, 0, 0, 0',
	X =  1507.182  mm,	Y =     4.462  mm,	Z =   -40.845  mm,
	W =   -41.198 deg,	P =   -19.963 deg,	R =    73.684 deg
   GP2:
	UF : 0, UT : 1,
	J1=    90.000 deg,	J2=   -90.000 deg
};
P[1011]{
   GP1:
	UF : 1, UT : 1,		CONFIG : 'N U T, 0, 0, 0',
	X =  1502.545  mm,	Y =    19.573  mm,	Z =   -37.702  mm,
	W =   -32.690 deg,	P =   -32.825 deg,	R =    84.377 deg
   GP2:
	UF : 0, UT : 1,
	J1=    90.000 deg,	J2=   -90.000 deg
};
P[1012]{
   GP1:
	UF : 1, UT : 1,		CONFIG : 'N U T, 0, 0, 0',
	X =  1491.160  mm,	Y =    23.880  mm,	Z =   -39.934  mm,
	W =    -8.358 deg,	P =   -44.371 deg,	R =    89.878 deg
   GP2:
	UF : 0, UT : 1,
	J1=    90.000 deg,	J2=   -90.000 deg
};
P[1013]{
   GP1:
	UF : 1, UT : 1,		CONFIG : 'N U T, 0, 0, 0',
	X =  1465.449  mm,	Y =    30.534  mm,	Z =   -41.739  mm,
	W =    -8.375 deg,	P =   -44.374 deg,	R =    89.894 deg
   GP2:
	UF : 0, UT : 1,
	J1=    90.000 deg,	J2=   -90.000 deg
};
P[1014]{
   GP1:
	UF : 1, UT : 1,		CONFIG : 'N U T, 0, 0, 0',
	X =  1230.526  mm,	Y =  -235.159  mm,	Z =   238.096  mm,
	W =    25.573 deg,	P =   -37.026 deg,	R =    45.674 deg
   GP2:
	UF : 0, UT : 1,
	J1=    90.000 deg,	J2=   -90.000 deg
};
P[1015]{
   GP1:
	UF : 1, UT : 1,		CONFIG : 'N U T, 0, 0, 0',
	X =   933.242  mm,	Y =   221.976  mm,	Z =    97.147  mm,
	W =    34.687 deg,	P =    17.432 deg,	R =    80.127 deg
   GP2:
	UF : 0, UT : 1,
	J1=    90.000 deg,	J2=   -90.000 deg
};
P[1016]{
   GP1:
	UF : 1, UT : 1,		CONFIG : 'N U T, 0, 0, 0',
	X =  1695.711  mm,	Y =   392.370  mm,	Z =    51.456  mm,
	W =   -31.968 deg,	P =    31.913 deg,	R =   -49.728 deg
   GP2:
	UF : 0, UT : 1,
	J1=    90.000 deg,	J2=   -90.000 deg
};
P[1017]{
   GP1:
	UF : 1, UT : 1,		CONFIG : 'N U T, 0, 0, 0',
	X =  1681.017  mm,	Y =   491.023  mm,	Z =   -42.111  mm,
	W =   -27.131 deg,	P =    36.937 deg,	R =   -46.225 deg
   GP2:
	UF : 0, UT : 1,
	J1=    90.000 deg,	J2=   -90.000 deg
};
P[1018]{
   GP1:
	UF : 1, UT : 1,		CONFIG : 'N U T, 0, 0, 0',
	X =  1615.991  mm,	Y =    27.362  mm,	Z =   -42.588  mm,
	W =   -41.512 deg,	P =    19.281 deg,	R =   -77.925 deg
   GP2:
	UF : 0, UT : 1,
	J1=    90.000 deg,	J2=   -90.000 deg
};
P[1019]{
   GP1:
	UF : 1, UT : 1,		CONFIG : 'N U T, 0, 0, 0',
	X =  1698.143  mm,	Y =   167.061  mm,	Z =    99.809  mm,
	W =   -40.772 deg,	P =    18.032 deg,	R =   -44.164 deg
   GP2:
	UF : 0, UT : 1,
	J1=    90.000 deg,	J2=   -90.000 deg
};
P[1020]{
   GP1:
	UF : 1, UT : 1,		CONFIG : 'N U T, 0, 0, 0',
	X =  1908.299  mm,	Y =    54.865  mm,	Z =   113.676  mm,
	W =    42.650 deg,	P =   -11.738 deg,	R =  -106.796 deg
   GP2:
	UF : 0, UT : 1,
	J1=    75.000 deg,	J2=   -90.000 deg
};
P[1021]{
   GP1:
	UF : 1, UT : 1,		CONFIG : 'N U T, 0, 0, 0',
	X =  1953.951  mm,	Y =     5.632  mm,	Z =    39.145  mm,
	W =    29.608 deg,	P =   -16.799 deg,	R =  -110.643 deg
   GP2:
	UF : 0, UT : 1,
	J1=    75.000 deg,	J2=   -90.000 deg
};
P[1022]{
   GP1:
	UF : 1, UT : 1,		CONFIG : 'N U T, 0, 0, 0',
	X =  2027.889  mm,	Y =   108.049  mm,	Z =    16.247  mm,
	W =    31.674 deg,	P =   -11.950 deg,	R =  -119.063 deg
   GP2:
	UF : 0, UT : 1,
	J1=    75.000 deg,	J2=   -90.000 deg
};
P[1023]{
   GP1:
	UF : 1, UT : 1,		CONFIG : 'N U T, 0, 0, 0',
	X =  2038.465  mm,	Y =   126.921  mm,	Z =    16.472  mm,
	W =    31.104 deg,	P =   -20.985 deg,	R =  -124.826 deg
   GP2:
	UF : 0, UT : 1,
	J1=    75.000 deg,	J2=   -90.000 deg
};
P[1024]{
   GP1:
	UF : 1, UT : 1,		CONFIG : 'N U T, 0, 0, 0',
	X =  2054.929  mm,	Y =   139.425  mm,	Z =    12.702  mm,
	W =    20.533 deg,	P =   -35.689 deg,	R =  -113.476 deg
   GP2:
	UF : 0, UT : 1,
	J1=    75.000 deg,	J2=   -90.000 deg
};
P[1025]{
   GP1:
	UF : 1, UT : 1,		CONFIG : 'N U T, 0, 0, 0',
	X =  2359.489  mm,	Y =   285.327  mm,	Z =   -65.577  mm,
	W =     8.217 deg,	P =   -39.758 deg,	R =   -93.501 deg
   GP2:
	UF : 0, UT : 1,
	J1=    75.000 deg,	J2=   -90.000 deg
};
P[1026]{
   GP1:
	UF : 1, UT : 1,		CONFIG : 'N U T, 0, 0, 0',
	X =  2384.280  mm,	Y =   299.923  mm,	Z =   -71.556  mm,
	W =    18.277 deg,	P =   -31.096 deg,	R =   -91.382 deg
   GP2:
	UF : 0, UT : 1,
	J1=    75.000 deg,	J2=   -90.000 deg
};
P[1027]{
   GP1:
	UF : 1, UT : 1,		CONFIG : 'N U T, 0, 0, 0',
	X =  2405.415  mm,	Y =   321.632  mm,	Z =   -77.444  mm,
	W =    10.697 deg,	P =   -31.045 deg,	R =   -61.018 deg
   GP2:
	UF : 0, UT : 1,
	J1=    75.000 deg,	J2=   -90.000 deg
};
P[1028]{
   GP1:
	UF : 1, UT : 1,		CONFIG : 'N U T, 0, 0, 0',
	X =  2518.007  mm,	Y =   526.725  mm,	Z =  -104.573  mm,
	W =    -9.006 deg,	P =   -31.541 deg,	R =   -24.015 deg
   GP2:
	UF : 0, UT : 1,
	J1=    75.000 deg,	J2=   -90.000 deg
};
P[1029]{
   GP1:
	UF : 1, UT : 1,		CONFIG : 'N U T, 0, 0, 0',
	X =  2529.887  mm,	Y =   547.837  mm,	Z =  -109.688  mm,
	W =     1.676 deg,	P =   -30.642 deg,	R =   -24.071 deg
   GP2:
	UF : 0, UT : 1,
	J1=    74.999 deg,	J2=   -90.000 deg
};
P[1030]{
   GP1:
	UF : 1, UT : 1,		CONFIG : 'N U T, 0, 0, 0',
	X =  2532.521  mm,	Y =   570.458  mm,	Z =  -110.392  mm,
	W =    11.600 deg,	P =   -27.859 deg,	R =   -23.691 deg
   GP2:
	UF : 0, UT : 1,
	J1=    75.000 deg,	J2=   -90.000 deg
};
P[1031]{
   GP1:
	UF : 1, UT : 1,		CONFIG : 'N U T, 0, 0, 0',
	X =  2532.281  mm,	Y =   890.860  mm,	Z =  -109.269  mm,
	W =    11.580 deg,	P =   -27.866 deg,	R =   -23.681 deg
   GP2:
	UF : 0, UT : 1,
	J1=    75.000 deg,	J2=   -90.000 deg
};
P[1032]{
   GP1:
	UF : 1, UT : 1,		CONFIG : 'N U T, 0, 0, 0',
	X =  2420.365  mm,	Y =   890.931  mm,	Z =    73.687  mm,
	W =    11.586 deg,	P =   -27.867 deg,	R =   -23.683 deg
   GP2:
	UF : 0, UT : 1,
	J1=    75.000 deg,	J2=   -90.000 deg
};
P[1033]{
   GP1:
	UF : 1, UT : 1,		CONFIG : 'N U T, 0, 0, 0',
	X =  2354.334  mm,	Y =  1101.931  mm,	Z =    73.687  mm,
	W =    11.586 deg,	P =   -27.867 deg,	R =   -23.683 deg
   GP2:
	UF : 0, UT : 1,
	J1=    75.000 deg,	J2=   -90.000 deg
};
P[1034]{
   GP1:
	UF : 1, UT : 1,		CONFIG : 'N U T, 0, 0, 0',
	X =  2408.252  mm,	Y =  1078.896  mm,	Z =   -76.528  mm,
	W =    11.605 deg,	P =   -27.850 deg,	R =   -23.703 deg
   GP2:
	UF : 0, UT : 1,
	J1=    75.000 deg,	J2=   -90.000 deg
};
P[1035]{
   GP1:
	UF : 1, UT : 1,		CONFIG : 'N U T, 0, 0, 0',
	X =  2409.979  mm,	Y =  1063.424  mm,	Z =   -77.389  mm,
	W =    11.606 deg,	P =   -27.847 deg,	R =   -23.707 deg
   GP2:
	UF : 0, UT : 1,
	J1=    75.000 deg,	J2=   -90.000 deg
};
P[1036]{
   GP1:
	UF : 1, UT : 1,		CONFIG : 'N U T, 0, 0, 0',
	X =  2414.410  mm,	Y =  1056.095  mm,	Z =   -80.691  mm,
	W =    34.423 deg,	P =     -.790 deg,	R =   -36.573 deg
   GP2:
	UF : 0, UT : 1,
	J1=    75.000 deg,	J2=   -90.000 deg
};
P[1037]{
   GP1:
	UF : 1, UT : 1,		CONFIG : 'N U T, 0, 0, 0',
	X =  2421.810  mm,	Y =  1053.185  mm,	Z =   -83.323  mm,
	W =    34.779 deg,	P =     -.071 deg,	R =   -37.103 deg
   GP2:
	UF : 0, UT : 1,
	J1=    75.000 deg,	J2=   -90.000 deg
};
P[1038]{
   GP1:
	UF : 1, UT : 1,		CONFIG : 'N U T, 0, 0, 0',
	X =  2438.564  mm,	Y =  1055.002  mm,	Z =   -88.542  mm,
	W =    45.658 deg,	P =    12.291 deg,	R =     2.752 deg
   GP2:
	UF : 0, UT : 1,
	J1=    75.000 deg,	J2=   -90.000 deg
};
P[1039]{
   GP1:
	UF : 1, UT : 1,		CONFIG : 'N U T, 0, 0, 0',
	X =  2488.520  mm,	Y =  1043.756  mm,	Z =  -101.823  mm,
	W =    40.993 deg,	P =    25.264 deg,	R =   -46.420 deg
   GP2:
	UF : 0, UT : 1,
	J1=    75.000 deg,	J2=   -90.000 deg
};
P[1040]{
   GP1:
	UF : 1, UT : 1,		CONFIG : 'N U T, 0, 0, 0',
	X =  2522.754  mm,	Y =  1010.208  mm,	Z =  -108.558  mm,
	W =    26.324 deg,	P =   -18.903 deg,	R =   -21.459 deg
   GP2:
	UF : 0, UT : 1,
	J1=    75.000 deg,	J2=   -90.000 deg
};
P[1041]{
   GP1:
	UF : 1, UT : 1,		CONFIG : 'N U T, 0, 0, 0',
	X =  2535.170  mm,	Y =   988.987  mm,	Z =  -111.768  mm,
	W =    32.199 deg,	P =   -12.971 deg,	R =   -18.013 deg
   GP2:
	UF : 0, UT : 1,
	J1=    75.000 deg,	J2=   -90.000 deg
};
P[1042]{
   GP1:
	UF : 1, UT : 1,		CONFIG : 'N U T, 0, 0, 0',
	X =  2546.209  mm,	Y =   956.342  mm,	Z =  -112.807  mm,
	W =    13.944 deg,	P =   -26.865 deg,	R =   -24.281 deg
   GP2:
	UF : 0, UT : 1,
	J1=    74.999 deg,	J2=   -90.000 deg
};
P[1043]{
   GP1:
	UF : 1, UT : 1,		CONFIG : 'N U T, 0, 0, 0',
	X =  2538.801  mm,	Y =   929.373  mm,	Z =  -111.510  mm,
	W =    -6.471 deg,	P =   -31.595 deg,	R =   -24.635 deg
   GP2:
	UF : 0, UT : 1,
	J1=    75.000 deg,	J2=   -90.000 deg
};
P[1044]{
   GP1:
	UF : 1, UT : 1,		CONFIG : 'N U T, 0, 0, 0',
	X =  2534.564  mm,	Y =   915.670  mm,	Z =  -110.094  mm,
	W =     1.523 deg,	P =   -30.709 deg,	R =   -24.701 deg
   GP2:
	UF : 0, UT : 1,
	J1=    75.000 deg,	J2=   -90.000 deg
};
P[1045]{
   GP1:
	UF : 1, UT : 1,		CONFIG : 'N U T, 0, 0, 0',
	X =  2533.629  mm,	Y =   887.767  mm,	Z =  -111.110  mm,
	W =    11.877 deg,	P =   -27.745 deg,	R =   -24.298 deg
   GP2:
	UF : 0, UT : 1,
	J1=    75.000 deg,	J2=   -90.000 deg
};
P[1046]{
   GP1:
	UF : 1, UT : 1,		CONFIG : 'N U T, 0, 0, 0',
	X =  2411.102  mm,	Y =   894.517  mm,	Z =    90.509  mm,
	W =    13.605 deg,	P =   -31.054 deg,	R =   -25.134 deg
   GP2:
	UF : 0, UT : 1,
	J1=    75.000 deg,	J2=   -90.000 deg
};
P[1047]{
   GP1:
	UF : 1, UT : 1,		CONFIG : 'N U T, 0, 0, 0',
	X =  2411.145  mm,	Y =   894.399  mm,	Z =   416.736  mm,
	W =    23.304 deg,	P =   -45.350 deg,	R =   -31.189 deg
   GP2:
	UF : 0, UT : 1,
	J1=    75.000 deg,	J2=   -90.000 deg
};
P[1048]{
   GP1:
	UF : 1, UT : 1,		CONFIG : 'N U T, 0, 0, 0',
	X =  1339.173  mm,	Y =   894.353  mm,	Z =   608.675  mm,
	W =    23.298 deg,	P =   -45.347 deg,	R =   -31.185 deg
   GP2:
	UF : 0, UT : 1,
	J1=    75.000 deg,	J2=   -90.000 deg
};
P[1049]{
   GP1:
	UF : 1, UT : 1,		CONFIG : 'N U T, 0, 0, 0',
	X =    97.559  mm,	Y =   894.331  mm,	Z =   608.685  mm,
	W =   -19.983 deg,	P =    41.209 deg,	R =   -28.759 deg
   GP2:
	UF : 0, UT : 1,
	J1=    75.000 deg,	J2=   -90.000 deg
};
P[1050]{
   GP1:
	UF : 1, UT : 1,		CONFIG : 'N U B, 0, 0, 0',
	X =   390.531  mm,	Y =    -9.911  mm,	Z =  2433.853  mm,
	W =     -.021 deg,	P =   -39.773 deg,	R =      .020 deg
   GP2:
	UF : 0, UT : 1,
	J1=    90.000 deg,	J2=   -90.000 deg
};
P[1051]{
   GP1:
	UF : 1, UT : 1,		CONFIG : 'N U T, 0, 0, 0',
	X =  2087.763  mm,	Y =  -128.190  mm,	Z =  1257.777  mm,
	W =     1.267 deg,	P =    49.420 deg,	R =  -164.947 deg
   GP2:
	UF : 0, UT : 1,
	J1=    89.999 deg,	J2=   -90.000 deg
};
P[1052]{
   GP1:
	UF : 1, UT : 1,		CONFIG : 'N U T, 0, 0, 0',
	X =  2078.822  mm,	Y =  -128.879  mm,	Z =   865.846  mm,
	W =     -.347 deg,	P =    42.653 deg,	R =  -165.506 deg
   GP2:
	UF : 0, UT : 1,
	J1=    89.999 deg,	J2=   -90.000 deg
};
P[1053]{
   GP1:
	UF : 1, UT : 1,		CONFIG : 'N U T, 0, 0, 0',
	X =  2063.478  mm,	Y =   -90.278  mm,	Z =   868.406  mm,
	W =     -.673 deg,	P =    43.750 deg,	R =  -163.703 deg
   GP2:
	UF : 0, UT : 1,
	J1=    89.999 deg,	J2=   -90.000 deg
};
P[1054]{
   GP1:
	UF : 1, UT : 1,		CONFIG : 'N U T, 0, 0, 0',
	X =  2042.660  mm,	Y =   -80.120  mm,	Z =   864.230  mm,
	W =     -.886 deg,	P =    43.217 deg,	R =   -85.673 deg
   GP2:
	UF : 0, UT : 1,
	J1=    89.999 deg,	J2=   -90.000 deg
};
P[1055]{
   GP1:
	UF : 1, UT : 1,		CONFIG : 'N U T, 0, 0, 0',
	X =  2029.699  mm,	Y =   -99.089  mm,	Z =   862.541  mm,
	W =     -.858 deg,	P =    43.081 deg,	R =    13.456 deg
   GP2:
	UF : 0, UT : 1,
	J1=    90.000 deg,	J2=   -90.000 deg
};
P[1056]{
   GP1:
	UF : 1, UT : 1,		CONFIG : 'N U T, 0, 0, 0',
	X =  2044.764  mm,	Y =  -145.522  mm,	Z =   863.704  mm,
	W =     -.844 deg,	P =    43.074 deg,	R =    16.885 deg
   GP2:
	UF : 0, UT : 1,
	J1=    90.000 deg,	J2=   -90.000 deg
};
P[1057]{
   GP1:
	UF : 1, UT : 1,		CONFIG : 'N U T, 0, 0, 0',
	X =  2066.345  mm,	Y =  -156.599  mm,	Z =   862.610  mm,
	W =     -.954 deg,	P =    42.968 deg,	R =   105.667 deg
   GP2:
	UF : 0, UT : 1,
	J1=    89.999 deg,	J2=   -90.000 deg
};
P[1058]{
   GP1:
	UF : 1, UT : 1,		CONFIG : 'N U T, 0, 0, 1',
	X =  2081.369  mm,	Y =  -128.535  mm,	Z =   863.747  mm,
	W =      .008 deg,	P =    43.052 deg,	R =  -165.933 deg
   GP2:
	UF : 0, UT : 1,
	J1=    89.999 deg,	J2=   -90.000 deg
};
P[1059]{
   GP1:
	UF : 1, UT : 1,		CONFIG : 'N U T, 0, 0, 0',
	X =  2038.233  mm,	Y =  -145.751  mm,	Z =  1040.502  mm,
	W =    -2.503 deg,	P =    37.782 deg,	R =  -167.602 deg
   GP2:
	UF : 0, UT : 1,
	J1=    90.000 deg,	J2=   -90.000 deg
};
P[1060]{
   GP1:
	UF : 1, UT : 1,		CONFIG : 'N U T, 0, 0, 0',
	X =  2074.921  mm,	Y =  -215.408  mm,	Z =  1040.502  mm,
	W =    -2.060 deg,	P =    34.855 deg,	R =   -96.844 deg
   GP2:
	UF : 0, UT : 1,
	J1=    90.000 deg,	J2=   -90.000 deg
};
P[1061]{
   GP1:
	UF : 1, UT : 1,		CONFIG : 'N U T, 0, 0, 0',
	X =  2058.688  mm,	Y =  -186.676  mm,	Z =   863.698  mm,
	W =    -3.996 deg,	P =    46.116 deg,	R =   -98.098 deg
   GP2:
	UF : 0, UT : 1,
	J1=    90.000 deg,	J2=   -90.000 deg
};
P[1062]{
   GP1:
	UF : 1, UT : 1,		CONFIG : 'N U T, 0, 0, 0',
	X =  2173.700  mm,	Y =  -185.156  mm,	Z =   864.180  mm,
	W =    -3.996 deg,	P =    46.103 deg,	R =   -98.114 deg
   GP2:
	UF : 0, UT : 1,
	J1=    90.000 deg,	J2=   -90.000 deg
};
P[1063]{
   GP1:
	UF : 1, UT : 1,		CONFIG : 'N U T, 0, 0, 0',
	X =  2223.219  mm,	Y =  -162.280  mm,	Z =   864.075  mm,
	W =    -3.959 deg,	P =    46.138 deg,	R =   -62.981 deg
   GP2:
	UF : 0, UT : 1,
	J1=    90.000 deg,	J2=   -90.000 deg
};
P[1064]{
   GP1:
	UF : 1, UT : 1,		CONFIG : 'N U T, 0, 0, 0',
	X =  2244.813  mm,	Y =  -121.390  mm,	Z =   863.141  mm,
	W =    -3.944 deg,	P =    46.113 deg,	R =   -22.988 deg
   GP2:
	UF : 0, UT : 1,
	J1=    90.000 deg,	J2=   -90.000 deg
};
P[1065]{
   GP1:
	UF : 1, UT : 1,		CONFIG : 'N U T, 0, 0, 0',
	X =  2359.031  mm,	Y =    58.406  mm,	Z =   866.058  mm,
	W =    -3.994 deg,	P =    46.113 deg,	R =   -65.223 deg
   GP2:
	UF : 0, UT : 1,
	J1=    90.000 deg,	J2=   -90.000 deg
};
P[1066]{
   GP1:
	UF : 1, UT : 1,		CONFIG : 'N U T, 0, 0, 0',
	X =  2555.017  mm,	Y =    95.013  mm,	Z =   866.214  mm,
	W =    -4.002 deg,	P =    46.108 deg,	R =  -103.330 deg
   GP2:
	UF : 0, UT : 1,
	J1=    90.000 deg,	J2=   -90.000 deg
};
P[1067]{
   GP1:
	UF : 1, UT : 1,		CONFIG : 'N U T, 0, 0, 0',
	X =  2606.669  mm,	Y =   110.131  mm,	Z =   866.023  mm,
	W =    11.847 deg,	P =    45.031 deg,	R =   -52.693 deg
   GP2:
	UF : 0, UT : 1,
	J1=    90.000 deg,	J2=   -90.000 deg
};
P[1068]{
   GP1:
	UF : 1, UT : 1,		CONFIG : 'N U T, 0, 0, 0',
	X =  2623.054  mm,	Y =   132.544  mm,	Z =   866.749  mm,
	W =    36.071 deg,	P =    31.153 deg,	R =    10.129 deg
   GP2:
	UF : 0, UT : 1,
	J1=    90.000 deg,	J2=   -90.000 deg
};
P[1069]{
   GP1:
	UF : 1, UT : 1,		CONFIG : 'N U T, 0, 0, 0',
